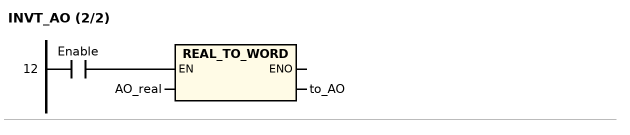
// NETWORK 12
IF Enable THEN to_AO := REAL_TO_WORD(AO_real); END_IF

END_FUNCTION_BLOCK

// Device/Application/Alarm
FUNCTION_BLOCK Alarm
VAR
	hw_alarm: STRING;
	R_DI121: R_TRIG;
	R_DI122: R_TRIG;
	R_DI123: R_TRIG;
	R_DI124: R_TRIG;
	R_DI125: R_TRIG;
	R_DI126: R_TRIG;
	R_DI127: R_TRIG;
	R_DI128: R_TRIG;
	
	B_DI121: INT;
	B_DI122: INT;
	B_DI123: INT;
	B_DI124: INT;
	B_DI125: INT;
	B_DI126: INT;
	B_DI127: INT;
	B_DI128: INT;
	
	R_DI131: R_TRIG;
	R_DI132: R_TRIG;
	R_DI133: R_TRIG;
	R_DI134: R_TRIG;
	R_DI135: R_TRIG;
	R_DI136: R_TRIG;
	R_DI137: R_TRIG;
	
	R_DI156: R_TRIG;
	
	R_DI162: R_TRIG;
	R_DI164: R_TRIG;
	R_DI166: R_TRIG;
	
	R_DI171: R_TRIG;
	R_DI172: R_TRIG;
	R_DI173: R_TRIG;
	R_DI174: R_TRIG;
	
	R_DI178: R_TRIG;
	
	R_DI181: R_TRIG;
	R_DI182: R_TRIG;
	R_DI183: R_TRIG;
	R_DI184: R_TRIG;
	R_DI185: R_TRIG;
	R_DI186: R_TRIG;
	R_DI187: R_TRIG;
	R_DI188: R_TRIG;
	
	R_DI191: R_TRIG;
	R_DI192: R_TRIG;
	R_DI193: R_TRIG;
	R_DI194: R_TRIG;
	R_DI195: R_TRIG;
	R_DI196: R_TRIG;
	
	R_DI201: R_TRIG;
	R_DI207: R_TRIG;
	R_DI208: R_TRIG;
	
	R_DI211: R_TRIG;
	
	R_DI221: R_TRIG;
	
	R_DI238: R_TRIG;
	
	R_DI241: R_TRIG;
	R_DI247: R_TRIG;
	R_DI248: R_TRIG;
	
	R_DI251: R_TRIG;
	
	alarm_ar: INT;
END_VAR

R_DI121(CLK:= DI121, Q=> );
R_DI122(CLK:= DI122, Q=> );
R_DI123(CLK:= DI123, Q=> );
R_DI124(CLK:= DI124, Q=> );
R_DI125(CLK:= DI125, Q=> );
R_DI126(CLK:= DI126, Q=> );
R_DI127(CLK:= DI127, Q=> );
R_DI128(CLK:= DI128, Q=> );
IF R_DI121.Q = TRUE AND alarm_ar < 40 THEN
	alarm_ar := alarm_ar + 1;
	hw_alarm := 'Q21 Vibrator 1 Cement Silo TRIP';
	B_DI121 := alarm_ar;
END_IF
IF R_DI122.Q = TRUE AND alarm_ar < 40 THEN
	alarm_ar := alarm_ar + 1;
	hw_alarm := 'Q23 Vibrator 2 Cement Silo TRIP';
	B_DI122 := alarm_ar; 
END_IF
IF R_DI123.Q = TRUE AND alarm_ar < 40 THEN
	alarm_ar := alarm_ar + 1;
	hw_alarm := 'Q25 Rotary Cement Silo TRIP';
	B_DI123 := alarm_ar; 
END_IF
IF R_DI124.Q = TRUE AND alarm_ar < 40 THEN
	alarm_ar := alarm_ar + 1;
	hw_alarm := 'Q27 Rotary Cement Weighter TRIP';
	B_DI124 := alarm_ar; 
END_IF
IF R_DI125.Q = TRUE AND alarm_ar < 40 THEN
	alarm_ar := alarm_ar + 1;
	hw_alarm := 'Q21 Vibrator 1 Cement Silo TRIP';
	B_DI125 := alarm_ar; 
END_IF
IF R_DI126.Q = TRUE AND alarm_ar < 40 THEN
	alarm_ar := alarm_ar + 1;
	hw_alarm := 'Q21 Vibrator 1 Cement Silo TRIP';
	B_DI126 := alarm_ar; 
END_IF
IF R_DI127.Q = TRUE AND alarm_ar < 40 THEN
	alarm_ar := alarm_ar + 1;
	hw_alarm := 'Q21 Vibrator 1 Cement Silo TRIP';
	B_DI127 := alarm_ar; 
END_IF
IF R_DI128.Q = TRUE AND alarm_ar < 40 THEN
	alarm_ar := alarm_ar + 1;
	hw_alarm := 'Q21 Vibrator 1 Cement Silo TRIP';
	B_DI128 := alarm_ar; 
END_IF

END_FUNCTION_BLOCK

// Device/Application/Constancheck
FUNCTION_BLOCK Constancheck
VAR
	ton_a: ton;
	ton_b: ton;
	catcher: r_trig;
	buffer: REAL;
	up_limit: REAL;
	down_limit: REAL;
	valid: INT;
	start_cek: BOOL;
END_VAR
VAR_INPUT
	input_value: REAL;
	tolerance: REAL := 1;
	start: BOOL;
END_VAR

VAR_OUTPUT
	output: BOOL;
END_VAR

IF start = TRUE THEN
	valid := 0;
	start_cek := TRUE;
END_IF
ton_a(IN:= NOT ton_b.Q, PT:= T#100MS, Q=> , ET=> );
ton_b(IN:= ton_a.Q, PT:= T#100MS, Q=> , ET=> );
catcher(CLK:= ton_b.Q, Q=> );
IF catcher.Q = TRUE THEN
	buffer := input_value;
	up_limit := input_value + tolerance;
	down_limit := input_value - tolerance;
	IF buffer < up_limit AND buffer > down_limit THEN
		valid := valid + 1;
		ELSE
			valid := 0;
	END_IF
END_IF
IF valid >= 25 AND start_cek = TRUE THEN
	output := TRUE;
	start_cek := FALSE;
	ELSE
		output := FALSE;
END_IF

END_FUNCTION_BLOCK

// Device/Application/DC
FUNCTION_BLOCK DC
VAR
	TON_int1: TON;
	pulse_active: BOOL;
END_VAR
VAR_OUTPUT
	tmp_int: TIME;
END_VAR
VAR
	pulse_finish: BOOL;
	CTU_0: CTU;
	TON_pulse: TON;
	TON_distance: TON;
	tmp_pulse: TIME;
	valve: INT;
	distancing: BOOL;
	tmp_dis: TIME;
END_VAR
VAR_INPUT
	pulse: TIME;
	distance: TIME;
	valve_num: INT := 6;
END_VAR
VAR
	pulsing: BOOL;
END_VAR

VAR_INPUT
	interval: TIME;
END_VAR
VAR_OUTPUT
	out_signal: WORD;
END_VAR
VAR // added by the converter: edge detectors and wires of the graphical bodies
    _rt1, _rt2, _rt3, _rt4, _rt5 : R_TRIG;
    _w1 : BOOL;
END_VAR

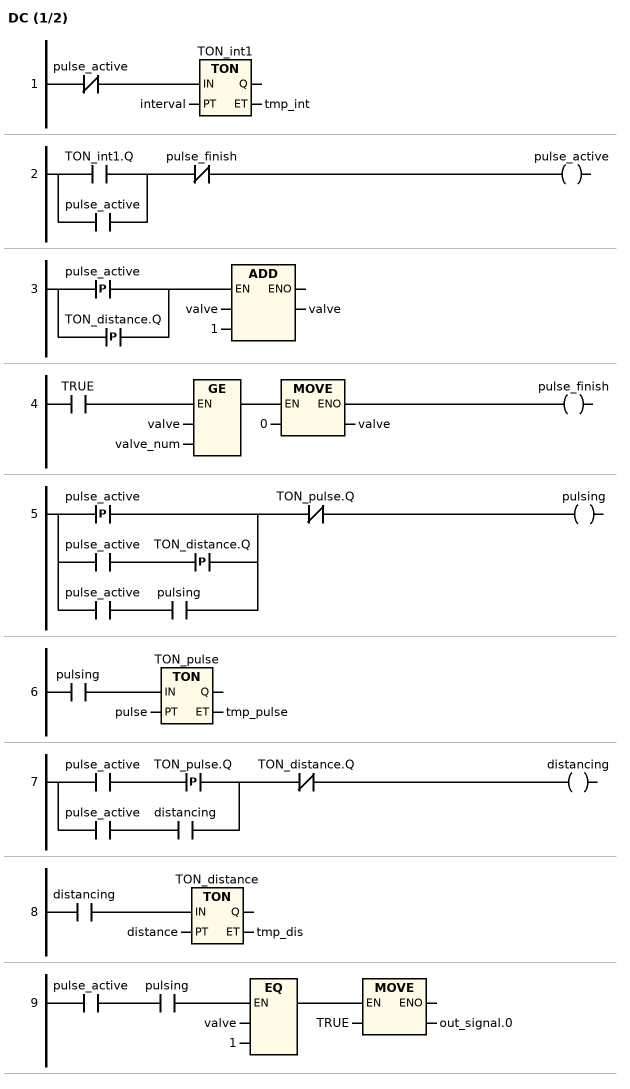
// NETWORK 1
TON_int1(IN := NOT pulse_active, PT := interval, ET => tmp_int); // TON

// NETWORK 2
pulse_active := (TON_int1.Q OR pulse_active) AND NOT pulse_finish;

// NETWORK 3
_rt1(CLK := pulse_active);
_rt2(CLK := TON_distance.Q);
IF _rt1.Q OR _rt2.Q THEN valve := valve + 1; END_IF

// NETWORK 4
_w1 := valve >= valve_num;
IF _w1 THEN valve := 0; END_IF
pulse_finish := _w1;

// NETWORK 5
_rt3(CLK := pulse_active);
_rt4(CLK := TON_distance.Q);
pulsing := (_rt3.Q OR pulse_active AND _rt4.Q OR pulse_active AND pulsing) AND NOT TON_pulse.Q;

// NETWORK 6
TON_pulse(IN := pulsing, PT := pulse, ET => tmp_pulse); // TON

// NETWORK 7
_rt5(CLK := TON_pulse.Q);
distancing := (pulse_active AND _rt5.Q OR pulse_active AND distancing) AND NOT TON_distance.Q;

// NETWORK 8
TON_distance(IN := distancing, PT := distance, ET => tmp_dis); // TON

// NETWORK 9
IF pulse_active AND pulsing AND valve = 1 THEN out_signal.0 := TRUE; END_IF

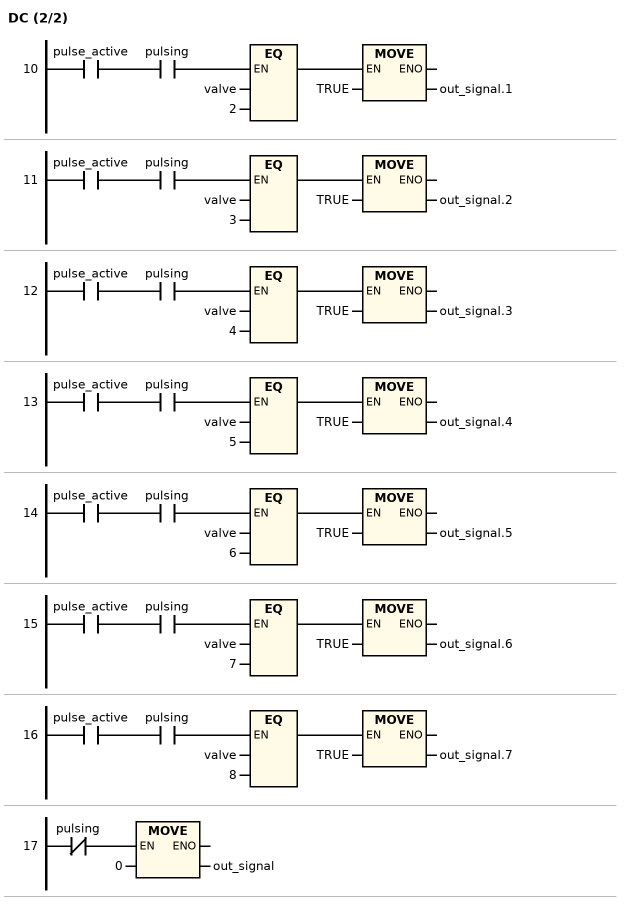
// NETWORK 10
IF pulse_active AND pulsing AND valve = 2 THEN out_signal.1 := TRUE; END_IF

// NETWORK 11
IF pulse_active AND pulsing AND valve = 3 THEN out_signal.2 := TRUE; END_IF

// NETWORK 12
IF pulse_active AND pulsing AND valve = 4 THEN out_signal.3 := TRUE; END_IF

// NETWORK 13
IF pulse_active AND pulsing AND valve = 5 THEN out_signal.4 := TRUE; END_IF

// NETWORK 14
IF pulse_active AND pulsing AND valve = 6 THEN out_signal.5 := TRUE; END_IF

// NETWORK 15
IF pulse_active AND pulsing AND valve = 7 THEN out_signal.6 := TRUE; END_IF

// NETWORK 16
IF pulse_active AND pulsing AND valve = 8 THEN out_signal.7 := TRUE; END_IF

// NETWORK 17
IF NOT pulsing THEN out_signal := 0; END_IF

END_FUNCTION_BLOCK

// Device/Application/PulseHold
FUNCTION_BLOCK PulseHold
VAR
	TON_PX : TON;
	pulse_in: BOOL;
	tmp_pulse: TIME;
	pulse_in2: BOOL;
END_VAR

VAR_INPUT
	sensor: BOOL;
	tolerance: TIME := T#5s;
	enable: BOOL;
END_VAR

VAR_OUTPUT
	output: BOOL;
END_VAR
VAR // added by the converter: edge detectors and wires of the graphical bodies
    _rt1 : R_TRIG;
    _ft1 : F_TRIG;
END_VAR

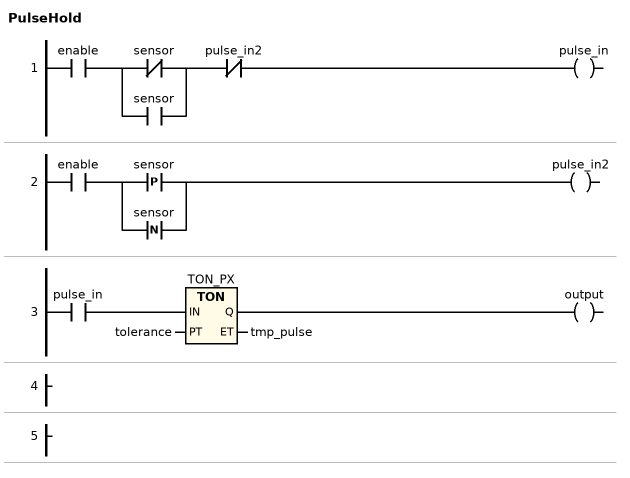
// NETWORK 1
pulse_in := enable AND (NOT sensor OR sensor) AND NOT pulse_in2;

// NETWORK 2
_rt1(CLK := sensor);
_ft1(CLK := sensor);
pulse_in2 := enable AND (_rt1.Q OR _ft1.Q);

// NETWORK 3
TON_PX(IN := pulse_in, PT := tolerance, ET => tmp_pulse); // TON
output := TON_PX.Q;

// NETWORK 4

// NETWORK 5

END_FUNCTION_BLOCK

// Device/Application/Logger
PROGRAM Logger
VAR
	oMySql : MySQL_Context; (* Used like Structure for keeping login and status information - Do not call it within your program *)
	
	
	(* Functionblock to contact MySql server *)
	
	oLogin : MYSQL_Login;
	xConnect : BOOL;
	diErrorLogin : DINT;
	sStatusLogin : STRING(200);
	xConnected : BOOL;

	(* Functionblock to process SQL statements who do not return result sets *)
	oExec1 : MYSQL_Execute;
	asSqlStatement1 : ARRAY [0..gcMySql_iSqlUpperBound] OF STRING(gcMySQL_iSqlLength);
	xExec1 : BOOL;
	diErrorExec1 : DINT;
	sStatusExec1 : STRING(200);

	(* Functionblock to process SQL statements who return result sets *)
	oQuery2 : MySQL_Query;
	asSqlStatement2 : ARRAY [0..gcMySql_iSqlUpperBound] OF STRING(gcMySQL_iSqlLength);
	xQuery2 : BOOL;
	diErrorQuery2 : DINT;
	sStatusQuery2 : STRING(200);
	stResultSet :MySQL_ResultSet;

	(* Functionblock to disconnect from MSSQL server *)
	oLogout : MySQL_Logout;
	xDisconnect : BOOL;
	diErrorLogout : DINT;
	sStatusLogout : STRING(200);

	
	TON_CONNECT: TON;
	
	TOF_RESETER: TOF;
	reseting: BOOL;
	res: R_TRIG;
END_VAR

TON_CONNECT( IN := NOT xConnected, PT := T#10S);
 
IF TON_CONNect.Q THEN 
	TON_CONNECT( IN := FALSE, PT := T#10S);
	xConnect := TRUE;
END_IF


oLogin(
	sHost:= '192.168.1.11', 
	uiPort:= 3306, 
	sUsername:= 'nodejs', 
	sPassword:= 'nodejs', 
	//sAppName:= , 
	//sLibName:= , 
	sDatabase:= 'db_codesys', 
	oMySql:= oMySql, 
	xStart:= xConnect, 
	diError=> diErrorLogin, 
	sStatus=> sStatusLogin, 
	xConnected=> xConnected);
	
	IF xConnected THEN
		IF Automode.log_mortar THEN 
			asSqlStatement1[0] := 'call mor(';
			asSqlStatement1[0] := CONCAT(asSqlStatement1[0], INT_TO_STRING(0));
			asSqlStatement1[0] := CONCAT(asSqlStatement1[0], ',"');
			asSqlStatement1[0] := CONCAT(asSqlStatement1[0], Formula.formula_name);
			asSqlStatement1[0] := CONCAT(asSqlStatement1[0], '",');
			asSqlStatement1[0] := CONCAT(asSqlStatement1[0], REAL_TO_STRING(Formula.cement_target));
			asSqlStatement1[0] := CONCAT(asSqlStatement1[0], ',');
			asSqlStatement1[0] := CONCAT(asSqlStatement1[0], REAL_TO_STRING(Formula.lime_target));
			asSqlStatement1[0] := CONCAT(asSqlStatement1[0], ',');
			asSqlStatement1[0] := CONCAT(asSqlStatement1[0], REAL_TO_STRING(Formula.sand_target));
			asSqlStatement1[0] := CONCAT(asSqlStatement1[0], ',');
			asSqlStatement1[0] := CONCAT(asSqlStatement1[0], REAL_TO_STRING(Automode.start_cement));
			asSqlStatement1[0] := CONCAT(asSqlStatement1[0], ',');
			asSqlStatement1[0] := CONCAT(asSqlStatement1[0], REAL_TO_STRING(Automode.end_cement));
			asSqlStatement1[0] := CONCAT(asSqlStatement1[0], ',');
			asSqlStatement1[0] := CONCAT(asSqlStatement1[0], INT_TO_STRING(Automode.weighting_duration));
			asSqlStatement1[0] := CONCAT(asSqlStatement1[0], ',');
			asSqlStatement1[0] := CONCAT(asSqlStatement1[0], REAL_TO_STRING(LimeSand.start_lime));
			asSqlStatement1[0] := CONCAT(asSqlStatement1[0], ',');
			asSqlStatement1[0] := CONCAT(asSqlStatement1[0], REAL_TO_STRING(LimeSand.end_lime));
			asSqlStatement1[0] := CONCAT(asSqlStatement1[0], ',');
			asSqlStatement1[0] := CONCAT(asSqlStatement1[0], INT_TO_STRING(LimeSand.weighting_duration));
			asSqlStatement1[0] := CONCAT(asSqlStatement1[0], ',');
			asSqlStatement1[0] := CONCAT(asSqlStatement1[0], REAL_TO_STRING(Cement_PRG.start_cement_dosing));
			asSqlStatement1[0] := CONCAT(asSqlStatement1[0], ',');
			asSqlStatement1[0] := CONCAT(asSqlStatement1[0], REAL_TO_STRING(Cement_PRG.end_cement_dosing));
			asSqlStatement1[0] := CONCAT(asSqlStatement1[0], ',');
			asSqlStatement1[0] := CONCAT(asSqlStatement1[0], INT_TO_STRING(Cement_PRG.dosing_duration));
			asSqlStatement1[0] := CONCAT(asSqlStatement1[0], ')');
			xExec1 := TRUE;
		END_IF
		IF LimeSand.finish_button THEN 
			asSqlStatement1[0] := 'INSERT INTO mo_lime(val, frm, act) VALUES(';
			asSqlStatement1[0] := CONCAT(asSqlStatement1[0], REAL_TO_STRING(LimeSand.lime_progress));
			asSqlStatement1[0] := CONCAT(asSqlStatement1[0], ',');
			asSqlStatement1[0] := CONCAT(asSqlStatement1[0], REAL_TO_STRING(Formula.lime_target));
			asSqlStatement1[0] := CONCAT(asSqlStatement1[0], ',');
			asSqlStatement1[0] := CONCAT(asSqlStatement1[0], REAL_TO_STRING(LimeSand.lime_weight));
			asSqlStatement1[0] := CONCAT(asSqlStatement1[0], ')');
			xExec1 := TRUE;
		END_IF
		IF Cement_PRG.log_cem THEN 
			asSqlStatement1[0] := 'INSERT INTO mo_cem(val, frm) VALUES(';
			asSqlStatement1[0] := CONCAT(asSqlStatement1[0], REAL_TO_STRING(Cement_PRG.cement_weight));
			asSqlStatement1[0] := CONCAT(asSqlStatement1[0], ',');
			asSqlStatement1[0] := CONCAT(asSqlStatement1[0], REAL_TO_STRING(formula.cement_target));
			asSqlStatement1[0] := CONCAT(asSqlStatement1[0], ')');
			xExec1 := TRUE;
		END_IF
		IF Automode.TON_4.Q THEN 
			asSqlStatement1[0] := 'INSERT INTO mo_clk(val) VALUES(';
			asSqlStatement1[0] := CONCAT(asSqlStatement1[0], '1');
			asSqlStatement1[0] := CONCAT(asSqlStatement1[0], ')');
			xExec1 := TRUE;
		END_IF
	END_IF
	
	
	oExec1(
	asSqlCommand:= asSqlStatement1, 
	oMySql:= oMySql, 
	xStart:= xExec1, 
	diError=> diErrorExec1, 
	sStatus=> sStatusExec1);
	
	IF diErrorExec1 <> 0 THEN
		reseting := TRUE;
	END_IF
	res(CLK:= reseting, Q=> );
	TOF_RESETER(IN:= res.Q, PT:= T#3S, Q=> , ET=> );

END_PROGRAM

// Device/Application/MYSQL/private/MySql_Context
FUNCTION_BLOCK MySql_Context
(*  This function block is used like a STRUCT for keeping login and status informations.
	
	Define one instance of this function block in your plc program and use it only as 
	input param for all the other function blocks of this library.

	Do not "call" this functionblock inside your plc program.

	In addition this function block provide the one and only receive and transmit buffer 
	for this library and operate as schedular for function blocks who want to talk with 
	the database server.
 *)
VAR_INPUT
  	sHost : STRING;		  	(* IP or hostname where MySQL-server is working *)
  	uiPort : UINT;			(* TCP-Port where MySQL-server is listening, typ. 3306 *)
	sUsername : STRING;
	sPassword : STRING;
	sDatabase : STRING;	  	(* Name of schema to use initially - Optional param*)

	stServerInfo : MySql_ServerInfo; (* See structure "MySql_ServerInfo" for details *)

	xConnected : BOOL; (* Succesful logged into database *)

	(*- Private ----------------------------------------------*)
	(* The one and only socket handle *)
	dwSocketHandle : DWORD; (* Handle for Read/Write data *)
	(* The one and only transmit buffer *)
	abTxBuffer	   : ARRAY[0..gcMySql_dwTxBufferSize] OF BYTE;
	(* The one and only receive buffer *)
	abRxBuffer	   : ARRAY[0..gcMySql_dwRxBufferSize] OF BYTE;
	(* The one and only semaphore to synchronize buffer access *)
	dwBufferSemaphor : DWORD; (* Handle to semaphore *)

END_VAR
VAR_OUTPUT
END_VAR
VAR

END_VAR

;

END_FUNCTION_BLOCK

// Device/Application/MYSQL/public/MySql_Login
FUNCTION_BLOCK MySql_Login
(* This function is used to connect to a MySQL-Server

	RetVal dwError:	
		16#00000000 => 'SUCCESS'
		16#80001001 => 'TCP-ERROR: DNS-Request failed, could not retrieve servers IP address'
		16#80001002 => 'TCP-ERROR: Could not convert servers IP address into dotted format'
		16#80001003 => 'TCP-ERROR: "SysSockCreate()" fails - Could not get socket'
		16#80001004 => 'TCP-ERROR: Switching to none blocking mode fails'
		16#80001005 => 'TCP-ERROR: "SysSockRecv()" returns 0. Socket was "gracefully closed"'
		16#80001006 => 'TCP-ERROR: "SysSockSend()" returns 0. Socket was "gracefully closed"'
		16#80001007 => 'TCP-ERROR: "SysSockSend()" returns -1'
		16#80004001 => 'PARAM-ERROR: ' 
		16#80004002 => 'PARAM-ERROR: "MySql.sHost" not assigned' 
		16#80004003 => 'PARAM-ERROR: "MySql.sUser" not assigned' 
		16#80005001 => 'MYSQL-ERROR: Library requires protocol version 10 or above. Server support only version x' 
		16#80005002 => 'MYSQL-ERROR: <Message from server>	
		16#80005003 => 'MYSQL-ERROR: Invalid or unexpected response from server'
		16#80005004 => 'MYSQL-ERROR: Function "MySql_Scramble()" returns with error'

		16#80004001 => 'TIMEOUT: <actual processed step in state machine>'

	ToDo's: 
		- Add checks for Server-Status and Server-Capabilties in "wState=35"

 date     | release	| author  | Desc
----------+---------+------------------------------------------------------------
 24.01.12 |  3.4	| CM      | Bugfix - Set PUSH-Bit also for 88x controllers 
 29.09.10 |  2.4    | CM      | Bugfix for IP in dotted format
 28.09.10 |  2.3    | CM      | Add DNS support for 750-881 and derivates
 28.09.10 |  2.2    | CM      | Add error message when Login not allowed for this host
 06.08.10 |  2.0	| CM      | Init 
*)
VAR_INPUT
  	sHost	  : STRING; 	 (* IP or hostname where MySQL-server is working *)
  	uiPort 	  : UINT := 3306;(* TCP-Port where MySQL-server is listening, typ. 3306 *)
	sUsername : STRING;		 (* Name of database account *)
	sPassword : STRING;   	 (* Password of database account *)
	sDatabase : STRING;	     (* Name of schema to use initially - Optional param*)
END_VAR
VAR_IN_OUT
	oMySql : MySql_Context;  (* Structure for keeping login and status informations *)
	xStart : BOOL; 			 (* Start execution on a rising edge and reset internally when done or on timeout.  *)
END_VAR
VAR_OUTPUT
	diError : DWORD; 		 (* Numeric return value - more readable in hex  *)
	sStatus : STRING(200); 	 (* Textual description of current state or error *)
	xConnected : BOOL;		 (* TRUE: when database connection is established *)
END_VAR
VAR
	wState : WORD;	 (* State mashine *)

	oTON			: TON;		(* Watchdogtimer for statemashine *)

	xWatchDogOn		: BOOL; 	(* enable disable Watchdog for statemashine *)
	wStateOld		: WORD;		(* persist the last state of statemashine *)

	sServerIpDotted	: STRING; 	(* Ip-Adress in dottet format '192.168.1.12' *)
	dwServerIp		: DWORD;	(* Ip-Adress in DWORD format  16#C0A8010C *)
	oInAddr	  		: INADDR;  	(* IP-Address as DWORD*)
	stSockAddr		: SOCKADDRESS;
	c_fdWrite : SOCKET_FD_SET;
	c_Timeout : SOCKET_TIMEVAL;

	dwSocket 	 	: DWORD; (* Socket handle *)
	diTcpOption  	: DINT := 1;
	diIoCtlParam 	: DINT := 1; (* IOCTL-Parameter for non-blocking mode of sockets *)
	xResult		 	: BOOL;		(* Return value of functions *)
	diResult		: __XINT; 	(* Retval value of functions *)

	diTxCount		: __XINT; (* Number of bytes to send *)
	diRxCount		: __XINT; (* Number of received bytes *)

	(* Local Buffer *)
	abToken : ARRAY[0..20] OF BYTE;  (* "abToken" calculatet from "salt" and "password" for login, when "password" is assigned *)

	(* Helpers *)
	dwPacketLength : DWORD; (*  *)
	uiPos : UINT;
	wMask : WORD := 16#00FF;
	dwMask : DWORD := 16#000000FF;

	i : INT;
	iHelp : INT;
	psHelp : POINTER TO STRING(180);
	pabHelp : POINTER TO ARRAY [0..512] OF BYTE;
	c_select: BOOL;
	RTS_IEC_RES: UDINT;
	ptrDINT : POINTER TO DINT;
	Sock_Host : SOCK_HOSTENT;
	Ready: INT;
	pIPAddress: POINTER TO DWORD;
END_VAR

CASE  wState OF (* The state maschine *********************************************)

0:	(* Idle - wait for something to do -------------------------------------------*)
	IF xStart THEN
		diError := 0;
		sStatus := '';
		MySql_Close(oMySql); (* Kill existing connection when user login two times *)
		oMySql.xConnected := FALSE;
		xConnected := oMySql.xConnected;
		wState := 5; (* Go ahead *)
	END_IF

5: (* Check structure "oMySql" for valid values *)
	IF sHost <> '' THEN
		oMySql.sHost := sHost;
	ELSE
		diError := 16#80004002;
		sStatus :='PARAM-ERROR: "sHost" not assigned';
		wState:=999;
		RETURN; (* ---- RETURN -----*)
	END_IF
	IF sUsername <> '' THEN
		oMySql.sUsername := sUsername;
	ELSE
		diError := 16#80004003;
		sStatus :='PARAM-ERROR: "sUsername" not assigned';
		wState:=999;
		RETURN; (* ---- RETURN -----*)
	END_IF
	oMySql.uiPort := uiPort;
	oMySql.sPassword := sPassword;
	oMySql.sDatabase := sDatabase;
	wState := 10; (* Go ahead *)

10:	(* Check if given address is "hostname" or "IP address in dottet format" --------------*)
	RTS_IEC_RES := SysSockInetAddr(oMySql.sHost, ADR(dwServerIp));
	IF RTS_IEC_RES = 16#00000000 AND dwServerIp <> 16#00000000 THEN
		sServerIpDotted:=oMySql.sHost;
		oInAddr.ulAddr := dwServerIp;
		wState:=15; 	(*Input is already the IP address in dottet format*)
	ELSE
		wState:=12; 	(*Input is a hostname *)
	END_IF

12: (* Send a DNS-Request to obtain servers IP address for the given hostname --------------*)
	RTS_IEC_RES := SysSockGetHostByName(oMySql.sHost,ADR(Sock_Host));
	pIPAddress := Sock_Host.pAddrList[0];
	dwServerIp := pIPAddress^;
	IF dwServerIp <> SOCKET_INADDR_NONE THEN
		wState:=14;
	ELSE
		diError := 16#80001001;
		sStatus :='TCP-ERROR: DNS-Request failed, could not retrieve servers IP address';
		wState:=999;
	END_IF

14: (* Convert Ip address from DWORD into dotted format ------------------------------------*)
(* Change byteorder from network to host order *)
	(*CASE ADR(%MW0) OF
	16#30000000 : (* For 750-841 *)
		oInAddr.S_addr:=SysSockNtohl(dwNet:=dwServerIp); (* Change byteorder from network to host order *)
	16#20000000 : (* For 750-881 *)
		oInAddr.S_addr:=SysSockNtohl(dwNet:=dwServerIp); (* Change byteorder from network to host order *)
	ELSE
		(* For 758-870 *)
		oInAddr.S_addr:= dwServerIp; (* Byteorder allready ok *)
	END_CASE*)
	oInAddr.ulAddr := dwServerIp; (* Byteorder allready ok *)
	RTS_IEC_RES := SysSockInetNtoa(pInAddr:=ADR(oInAddr), szIPAddr:= sServerIpDotted, diIPAddrSize:= SIZEOF(sServerIpDotted));
	xResult := (RTS_IEC_RES = 0);
	IF xResult THEN
		wState:=15;
	ELSE
		diError := 16#80001002;
		sStatus :='TCP-ERROR: Could not convert servers IP address into dotted format';
		wState:=999;
	END_IF

15: (* Create socket descriptor  ---------------------------*)
	(*dwSocket := SysSockCreate(diAddressFamily := SOCKET_AF_INET,
							  diType		  := SOCKET_STREAM,
							  diProtocol 	  := SOCKET_IPPROTO_IP);*)
	dwSocket := SysSockCreate(						 iAddressFamily	:= SOCKET_AF_INET,
													 diType		:= SOCKET_STREAM,
													 diProtocol := SOCKET_IPPROTO_TCP,
													 pResult := ADR(RTS_IEC_RES));
	IF dwSocket >= 0 THEN
		oMySql.dwSocketHandle := dwSocket;  (* Make handle available for other function blocks *)
		(* Set Push-Bit only for 750-841 and derivates *)
		IF TRUE THEN (*((ADR(%MW0)=16#30000000) OR (ADR(%MW0)=16#20000000)) THEN (*841, 871, 872, 873, 880 ... *)*)
			(*SysSockSetOption(diSocket		:= dwSocket,
							 diLevel		:= 6,
							 diOption		:= SOCKET_TCP_NODELAY,
							 pOptionValue	:= ADR(),
							 diOptionLength	:= SIZEOF(diTcpOption));*)
			SysSockSetOption(
						hSocket:=dwSocket,
						diLevel:=6,
						diOption:=SOCKET_TCP_NODELAY,
						pdiOptionValue:=ADR(diTcpOption),
						diOptionLen:=SIZEOF(diTcpOption));
		END_IF
		wState := 16; (* Go ahead *)
	ELSE
		diError := 16#80001003;
		sStatus :='TCP-ERROR: "SysSockCreate()" fails - Could not get socket';
		wState:=999;
	END_IF

16: (* Change socket mode to "nonblocking" ---------------------------*)
	diResult := SysSockIoctl( dwSocket,
							  SOCKET_FIONBIO,
							  ADR(diIoCtlParam));
	IF TRUE THEN (*diResult <> 0 THEN*)
		stSockAddr.sin_family := SOCKET_AF_INET;
		stSockAddr.sin_port := SysSockNtohs(uiPort);
		stSockAddr.sin_addr.ulAddr := oInAddr.ulAddr;
		sStatus := CONCAT('Try to connect with ', oMySql.sHost);
		wState := 18;
	ELSE
		diError := 16#80001004;
		sStatus :='TCP-ERROR: Switching to none blocking mode fails';
		wState:=999;
	END_IF

18: (* Create and occupy semaphore to synchronize buffer handling for socket operations *)
	oMySql.dwBufferSemaphor := SysSemCreate(ADR(RTS_IEC_RES)); (* Create semaphore  *)
	SysSemEnter(oMySql.dwBufferSemaphor); (* CAUTION: SysSemEnter() is a blocking function *)
	c_select := FALSE;
	wState := 20;

20: (* Connect with server ---------------------------*)
	sStatus :=CONCAT('Try to connect to ', oMySql.sHost);
	IF c_select = FALSE THEN
			RTS_IEC_RES := SysSockConnect( dwSocket, ADR(stSockAddr),  SIZEOF(stSockAddr));
			xResult := (RTS_IEC_RES = 0);
			IF NOT xResult THEN
						sStatus :='Connection established - Waiting for "Handshake Initialisation Packet" from server';
						wState:=25;
			ELSE
					c_select := TRUE;
			END_IF
	ELSE
			c_Timeout.tv_sec := 0;
			c_Timeout.tv_usec := 0;
			c_fdWrite.fd_count := 1;
			c_fdWrite.fd_array[0] := dwSocket;
			SysSockSelect(SOCKET_FD_SETSIZE,0,ADR(c_fdWrite),0, ADR(c_Timeout), ADR(Ready));
			xResult := Ready > 0;
			IF xResult THEN (* succesful *)
				sStatus :='Connection established - Waiting for "Handshake Initialisation Packet" from server';
				wState:=25;
			END_IF
	END_IF
25: (* Read "Handshake Initialisation Packet" received from server *)
	(*diRxCount := SysSockRecv(diSocket 	:= dwSocket,
							 pbyBuffer 	:= ADR(oMySql.abRxBuffer),		(* Address of receive buffer *)
							 diBufferSize:= SIZEOF(oMySql.abRxBuffer),
							 diFlags	:= 0);*)
		diRxCount := SysSockRecv(		hSocket 	:= dwSocket,
										pbyBuffer 	:= ADR(oMySql.abRxBuffer),		(* Address of receive buffer *)
										diBufferSize:= SIZEOF(oMySql.abRxBuffer),
										diFlags		:= 0,
										pResult := ADR(RTS_IEC_RES));						 

	CASE diRxCount OF
	-1:(* No data available or error occured *)
			; (* Let the watchdog look for *)

	(*0: (* Socket was "gracefully closed"  *)*)
		diError := 16#80001005;
		sStatus :='TCP-ERROR: "SysSockRecv()" returns 0. Socket was "gracefully closed"';
		wState:=999;

	ELSE (* We receive some data from server *)
		IF RTS_IEC_RES <> 0 AND RTS_IEC_RES <> 518 THEN
			diError := 16#80001005;
			sStatus :='TCP-ERROR: "SysSockRecv()" returns 0. Socket was "gracefully closed"';
			wState:=999;
		ELSE
		IF diRxCount > 0 THEN
		dwPacketLength := 	BYTE_TO_DWORD(oMySql.abRxBuffer[0]) OR
							SHL(BYTE_TO_DWORD(oMySql.abRxBuffer[1]),8) OR
							SHL(BYTE_TO_DWORD(oMySql.abRxBuffer[2]),16);
		IF diRxCount >= dwPacketLength THEN
			wState:=27; (* Go ahead *)
		END_IF
		END_IF
		END_IF
	END_CASE

27: (* Check if response a "Handshake Initialisation Packet" *)
	IF oMySql.abRxBuffer[4] = 16#FF THEN
		(* Error frame received - Copy error message *)
		psHelp := ADR(oMySql.abRxBuffer[7]);
		diError := 16#80005002;
		sStatus := CONCAT('MYSQL-ERROR: ', psHelp^);
		wState:=999;
	ELSE
		sStatus :='"Handshake Initialisation Packet" received - Generate "Scramble-Key"';
		wState:=30; (* Go ahead *)
	END_IF

30:	(* Copy informations from "server greetings" into context "oMySql.stServerInfo" *)
	(* Copy "Protocol-Version" to context *)
	oMySql.stServerInfo.bProtocolVersion := oMySql.abRxBuffer[4];
	(* Copy "Server-Version" to context *)
	psHelp := ADR(oMySql.abRxBuffer[5]);
	oMySql.stServerInfo.sServerVersion := psHelp^;
	(* Calculate Posion of Thread-Id in receive buffer *)
	uiPos := 5 +LEN(psHelp^)+1;
	(* Copy "Thread-Id"(4Byte) to context *)
	oMySql.stServerInfo.dwThreadId :=    BYTE_TO_DWORD(oMySql.abRxBuffer[uiPos])       OR
										SHL(BYTE_TO_DWORD(oMySql.abRxBuffer[uiPos+1]),8)  OR
										SHL(BYTE_TO_DWORD(oMySql.abRxBuffer[uiPos+2]),16) OR
										SHL(BYTE_TO_DWORD(oMySql.abRxBuffer[uiPos+3]),24);
	uiPos := uiPos +4;
	(* Copy first part (8Byte) of "Scramble-Buffer" to context *)
	FOR i:=0 TO 7 DO
		oMySql.stServerInfo.abScrambleBuffer[i] := oMySql.abRxBuffer[uiPos+i];
	END_FOR
	uiPos := uiPos +8 +1;
	(* Copy "Server-Capabilities" to context *)
	oMySql.stServerInfo.wServerCapabilities := 	BYTE_TO_WORD(oMySql.abRxBuffer[uiPos])       OR
												SHL(BYTE_TO_WORD(oMySql.abRxBuffer[uiPos+1]),8);
	uiPos := uiPos +2;
	(* Copy "Server-Language" to context *)
	oMySql.stServerInfo.bServerLanguageId := oMySql.abRxBuffer[uiPos];
	uiPos := uiPos +1;
	(* Copy "Server-Status" to context *)
	oMySql.stServerInfo.wServerStatus := BYTE_TO_WORD(oMySql.abRxBuffer[uiPos])       OR
										SHL(BYTE_TO_WORD(oMySql.abRxBuffer[uiPos+1]),8);
	uiPos := uiPos +2+13;
	(* Copy rest(13Byte) of "Scramble-Buffer" to context *)
	FOR i:=0 TO 12 DO
		oMySql.stServerInfo.abScrambleBuffer[8 +i] := oMySql.abRxBuffer[uiPos+i];
	END_FOR
	wState:=35;

35: (* Check informations from "server greetings" *)
	IF oMySql.stServerInfo.bProtocolVersion < 10 THEN
		diError := 16#80005001;
		sStatus :=CONCAT('MYSQL-ERROR: Library requires protocol version 10 or above. Server support only version ', BYTE_TO_STRING(oMySql.stServerInfo.bProtocolVersion));
		wState:=999;
		RETURN;
	END_IF
	wState:=40;

40: (* Calculate "Token" for login from "salt" and "password", when "password" is assigned *)
	IF oMySql.sPassword = '' THEN
		wState:=45;
	ELSE
		xResult := MySql_Scramble(oMySql.stServerInfo.abScrambleBuffer,
								  oMySql.sPassword,
							      abToken);
		IF xResult THEN
			wState:=45;
		ELSE
			diError := 16#80005004;
			sStatus :='MYSQL-ERROR: Function "MySql_Scramble()" returns with error';
			wState:=999;
		END_IF
	END_IF

45: (* Prepare "Client Authentication Packet" or "Login Request" ---------------------------*)
	(* Packet-Length - will be calculated and assigned at the end of this step *)
	oMySql.abTxBuffer[ 0] := 16#00;
	oMySql.abTxBuffer[ 1] := 16#00;
	oMySql.abTxBuffer[ 2] := 16#00;
	(* Packet-Number *)
	oMySql.abTxBuffer[ 3] := 1;
	(* Client-Capabilties *)
	oMySql.abTxBuffer[ 4] := WORD_TO_BYTE(gcMySql_wClientFlags AND wMask);
	oMySql.abTxBuffer[ 5] := WORD_TO_BYTE(SHR(gcMySql_wClientFlags, 8) AND wMask);
	(* Client-Capabilties - Extended *)
	oMySql.abTxBuffer[ 6] := WORD_TO_BYTE(gcMySql_wExtClientFlags AND wMask);
	oMySql.abTxBuffer[ 7] := WORD_TO_BYTE(SHR(gcMySql_wExtClientFlags, 8) AND wMask);
	(* Max-Packet-Size *)
	oMySql.abTxBuffer[ 8] := DWORD_TO_BYTE(gcMySql_dwMaxPacketSize AND dwMask);
	oMySql.abTxBuffer[ 9] := DWORD_TO_BYTE(SHR(gcMySql_dwMaxPacketSize, 8) AND dwMask);
	oMySql.abTxBuffer[10] := DWORD_TO_BYTE(SHR(gcMySql_dwMaxPacketSize, 16) AND dwMask);
	oMySql.abTxBuffer[11] := DWORD_TO_BYTE(SHR(gcMySql_dwMaxPacketSize, 24) AND dwMask);
	(* Character-Set *)
	oMySql.abTxBuffer[12] := gcMySql_bCharsetNumber;
	(* Filler - 23 byte allways 16#00 *)
	FOR i:=0 TO 22 DO
		oMySql.abTxBuffer[13+i] := 16#00;
	END_FOR
	uiPos := 13 + 23;
	(* Username (Null-Terminated String) *)
	pabHelp := ADR(sUsername);
	iHelp := LEN(sUsername);
	FOR i:=0 TO iHelp DO
		oMySql.abTxBuffer[uiPos+i] := pabHelp^[i];
	END_FOR
	uiPos := uiPos + iHelp +1;
	(* When Password is given *)
	IF sPassword = '' THEN
		(* Password (Length Coded Binary) *)
		oMySql.abTxBuffer[uiPos] := 16#00; (* Length *)
		uiPos := uiPos +1;
	ELSE
		(* Password (Length Coded Binary) *)
		oMySql.abTxBuffer[uiPos] := 20; (* Length *)
		uiPos := uiPos +1;
		(* Scrambled-Key *)
		FOR i:=0 TO 20 DO
			oMySql.abTxBuffer[uiPos+i] := abToken[i];
		END_FOR
		uiPos := uiPos +20;
	END_IF

	(* Calculate number of bytes to transmit and logical packet-length *)
	diTxCount := uiPos; (* Bytes to send *)
	dwPacketLength := uiPos -4;

	(* Packet-Length *)
	oMySql.abTxBuffer[ 0] := DWORD_TO_BYTE(dwPacketLength AND dwMask);
	oMySql.abTxBuffer[ 1] := DWORD_TO_BYTE(SHR(dwPacketLength, 8) AND dwMask);
	oMySql.abTxBuffer[ 2] := DWORD_TO_BYTE(SHR(dwPacketLength, 16) AND dwMask);
	sStatus :='Send "Login Request Packet" to server';
	wState := 50;

50: (* Send "Client Authentication Packet*)
	(*diResult := SysSockSend(diSocket := dwSocket,
							pbyBuffer := ADR(oMySql.abTxBuffer),
							diBufferSize := diTxCount,
							diFlags := 0);*)
	diResult := SysSockSend(	hSocket := dwSocket,
								pbyBuffer := ADR(oMySql.abTxBuffer),
								diBufferSize := diTxCount,
								diFlags := 0,
								pResult := ADR(RTS_IEC_RES));

	CASE diResult OF
	-1:	(* ERROR *)
		diError := 16#80001007;
		sStatus :='TCP-ERROR: "SysSockSend()" returns -1';
		wState:=999;
	0: (* Socket was "gracefully closed" *)
		diError := 16#80001007;
		sStatus :='TCP-ERROR: "SysSockSend()" returns 0. Socket was "gracefully closed"';
		wState:=999;
	ELSE (* succesful *)
		sStatus :='Waiting for "OK Packet" from server';
		wState:=55;
	END_CASE

55: (* Wait for "Response" from server *)
	(*diRxCount := SysSockRecv(diSocket 	:= dwSocket,
							 pbyBuffer 	:= ADR(oMySql.abRxBuffer),		(* Address of receive buffer *)
							 diBufferSize:= SIZEOF(oMySql.abRxBuffer),
							 diFlags	:= 0);*)
	diRxCount := SysSockRecv(		hSocket 	:= dwSocket,
										pbyBuffer 	:= ADR(oMySql.abRxBuffer),		(* Address of receive buffer *)
										diBufferSize:= SIZEOF(oMySql.abRxBuffer),
										diFlags		:= 0,
										pResult := ADR(RTS_IEC_RES));
	CASE diRxCount OF
	-1:(* No data available or error occured *)
			; (* Let the watchdog look for *)

	(*0: (* Socket was "gracefully closed"  *)*)
		diError := 16#80001005;
		sStatus :='TCP-ERROR: "SysSockRecv()" returns 0. Socket was "gracefully closed"';
		wState:=999;

	ELSE (* We receive some data from server *)
		IF RTS_IEC_RES <> 0 AND RTS_IEC_RES <> 518 THEN
			diError := 16#80001005;
			sStatus :='TCP-ERROR: "SysSockRecv()" returns 0. Socket was "gracefully closed"';
			wState:=999;
		ELSE
		IF diRxCount > 0 THEN
		dwPacketLength := 	BYTE_TO_DWORD(oMySql.abRxBuffer[0]) OR
							SHL(BYTE_TO_DWORD(oMySql.abRxBuffer[1]),8) OR
							SHL(BYTE_TO_DWORD(oMySql.abRxBuffer[2]),16);
		IF diRxCount >= dwPacketLength THEN
			wState:=60; (* Go ahead *)
		END_IF
		END_IF
		END_IF
	END_CASE

60: (* Check response packet, could be OK- or ERROR-Packet *)
	CASE oMySql.abRxBuffer[4] OF (* field "field_count"*)

	16#00: (* OK-Packet: Identified by "field_count", always = 0 *)
		IF sDatabase <> '' THEN
			(* Send "COM_INIT_DB" command to select specified database *)
			wState:=65;
		ELSE
			(* Everything fine - nothing else to do *)
			wState:=90;
		END_IF


	16#FF: (* ERROR-Packet: Identified by "field_count", always = 16#FF *)
		diError := 16#80005002;
		(* Copy server message into "sStatus"*)
		sStatus :='MYSQL-ERROR:  ';
		pabHelp := ADR(sStatus)+13;
		FOR i:=0 TO DWORD_TO_INT(dwPacketLength-10) DO
			pabHelp^[i] := oMySql.abRxBuffer[13+i];
			IF i>=499 THEN
				EXIT;
			END_IF
		END_FOR
		pabHelp^[i] := 16#00;
		wState:=999;

	ELSE (* Invalid or unexpected response from server (at this time) *)
		diError := 16#80005003;
		sStatus :='MYSQL-ERROR: Invalid or unexpected response from server';
		wState:=999;
	END_CASE

65: (* Prepare "COM_INIT_DB" command to select specified database *)
	(* Calculate Packet-Length *)
	iHelp := LEN(sDatabase); (* argument *)
	dwPacketLength := 1 + iHelp; (* command + argument *)
	diTxCount := dwPacketLength +4; (* Bytes to send (command + argument + header) *)
	(* Packet-Length *)
	oMySql.abTxBuffer[0] := DWORD_TO_BYTE(dwPacketLength AND dwMask);
	oMySql.abTxBuffer[1] := DWORD_TO_BYTE(SHR(dwPacketLength, 8) AND dwMask);
	oMySql.abTxBuffer[2] := DWORD_TO_BYTE(SHR(dwPacketLength, 16) AND dwMask);
	(* Packet-Number *)
	oMySql.abTxBuffer[3] := 0;
	(* Command *)
	oMySql.abTxBuffer[4] := 16#02; (* "COM_INIT_DB" command *)
	(* Argument *)
	pabHelp := ADR(sDatabase);
	FOR i:=0 TO iHelp-1 DO
		oMySql.abTxBuffer[5+i] := pabHelp^[i];
	END_FOR
 	(* Send "COM_INIT_DB" command to select specified database *)
	(*diResult := SysSockSend(diSocket := dwSocket,
							pbyBuffer := ADR(oMySql.abTxBuffer),
							diBufferSize := diTxCount,
							diFlags := 0);*)
	diResult := SysSockSend(	hSocket := dwSocket,
								pbyBuffer := ADR(oMySql.abTxBuffer),
								diBufferSize := diTxCount,
								diFlags := 0,
								pResult := ADR(RTS_IEC_RES));
							
	CASE diResult OF
	-1:	(* ERROR *)
		diError := 16#80001007;
		sStatus :='TCP-ERROR: "SysSockSend()" returns -1';
		wState:=999;
	0: (* Socket was "gracefully closed" *)
		diError := 16#80001007;
		sStatus :='TCP-ERROR: "SysSockSend()" returns 0. Socket was "gracefully closed"';
		wState:=999;
	ELSE (* succesful *)
		sStatus :='Waiting for "OK Packet" from server';
		wState:=70;
	END_CASE

70: (* Wait for "Response" from server *)
	(*diRxCount := SysSockRecv(diSocket 	:= dwSocket,
							 pbyBuffer 	:= ADR(oMySql.abRxBuffer),		(* Address of receive buffer *)
							 diBufferSize:= SIZEOF(oMySql.abRxBuffer),
							 diFlags	:= 0);*)
	diRxCount := SysSockRecv(			hSocket 	:= dwSocket,
										pbyBuffer 	:= ADR(oMySql.abRxBuffer),		(* Address of receive buffer *)
										diBufferSize:= SIZEOF(oMySql.abRxBuffer),
										diFlags		:= 0,
										pResult := ADR(RTS_IEC_RES));
	CASE diRxCount OF
	-1:(* No data available or error occured *)
			; (* Let the watchdog look for *)

	(*0: (* Socket was "gracefully closed"  *)*)
		diError := 16#80001005;
		sStatus :='TCP-ERROR: "SysSockRecv()" returns 0. Socket was "gracefully closed"';
		wState:=999;

	ELSE (* We receive some data from server *)
		IF RTS_IEC_RES <> 0 AND RTS_IEC_RES <> 518 THEN
			diError := 16#80001005;
			sStatus :='TCP-ERROR: "SysSockRecv()" returns 0. Socket was "gracefully closed"';
			wState:=999;
		ELSE
		IF diRxCount > 0 THEN
		dwPacketLength := 	BYTE_TO_DWORD(oMySql.abRxBuffer[0]) OR
							SHL(BYTE_TO_DWORD(oMySql.abRxBuffer[1]),8) OR
							SHL(BYTE_TO_DWORD(oMySql.abRxBuffer[2]),16);
		IF diRxCount >= dwPacketLength THEN
			wState:=75; (* Go ahead *)
		END_IF
		END_IF
		END_IF
	END_CASE

75: (* Check response packet, could be OK- or ERROR-Packet *)
	CASE oMySql.abRxBuffer[4] OF (* field "field_count"*)

	16#00: (* OK-Packet: Identified by "field_count", always = 0 *)
		wState:=90; (* Everything fine - nothing else to do *)

	16#FF: (* ERROR-Packet: Identified by "field_count", always = 16#FF *)
		diError := 16#80005002;
		(* Copy server message into "sStatus"*)
		sStatus :='MYSQL-ERROR:  ';
		pabHelp := ADR(sStatus)+13;
		FOR i:=0 TO DWORD_TO_INT(dwPacketLength-10) DO
			pabHelp^[i] := oMySql.abRxBuffer[13+i];
			IF i>=499 THEN
				EXIT;
			END_IF
		END_FOR
		pabHelp^[i] := 16#00;
		wState:=999;

	ELSE (* Invalid or unexpected response from server (at this time) *)
		diError := 16#80005003;
		sStatus :='MYSQL-ERROR: Invalid or unexpected response from server';
		wState:=999;
	END_CASE

90:	(* Connection established - Free semaphore to allow other function block access to Tx- and Rx-Buffer *)
	SysSemLeave(oMySql.dwBufferSemaphor);
	oMySql.xConnected := TRUE;
	xConnected := oMySql.xConnected;
	IF sDatabase = '' THEN
		sStatus := 'CONNECTED WITH DATABASE';
	ELSE
		sStatus := CONCAT('CONNECTED WITH DATABASE - "', sDatabase);
		sStatus := CONCAT(sStatus, '"');
	END_IF
	xStart := FALSE;
	wState:=100;

100: (* Wait here and check if socket is still alive *)
	IF oMySql.dwSocketHandle = 0 THEN
		xConnected := FALSE;
		sStatus := 'DISCONNECTED';
		wState:=999;
	END_IF
	IF xStart THEN
		wState := 0;
	END_IF

ELSE
	(* Clean up and close connection -----------------------------------------*)
	MySql_Close(oMySql); (* Kill existing connection *)
	xStart := FALSE;
	wState:=0;

END_CASE (**************************************************************************************)

(* Watchdog for statemachine  *)
IF oTON.Q THEN
	xWatchDogOn := FALSE;
	diError := 16#80004001; 	(* Watchdog time elapsed, see sStatus for details *)
	sStatus := CONCAT('TIMEOUT on:', sStatus);
	wState:=999;
END_IF

IF (wState > 0) AND (wState <> 100) THEN
	oTON(IN:=xWatchDogOn , PT:=gcMySql_tTimeOut);
	IF (wStateOld <> wState) THEN
		xWatchDogOn := FALSE; (* Step has changed *)
	ELSE
		xWatchDogOn := TRUE; (* Step still active *)
	END_IF
END_IF
wStateOld:=wState;

END_FUNCTION_BLOCK

// Device/Application/MYSQL/private/MySql_Close
FUNCTION MySql_Close : BOOL
(* This function closes database connection

	Do not "call" this function directly - Use function block "MySql_Logout" 
*)
VAR_IN_OUT
	oMySql : MySql_Context; (* Structure for keeping login and status informations *)
END_VAR
VAR
	i : INT;
END_VAR

IF oMySql.dwSocketHandle <> 0 THEN
	(* Call SysSockShutDown only for IPC's series 758-870  *)
	(*IF ((ADR(%MW0)=16#30000000) OR (ADR(%MW0)=16#20000000)) THEN (* 841 or 88x*)
		;
	ELSE*)
		SysSockShutdown(oMySql.dwSocketHandle, 0);(* 758-870 *)
	(*END_IF*)
	(* Call SysSockClose *)
	SysSockClose( oMySql.dwSocketHandle );
	(* Update context *)
	oMySql.dwSocketHandle := 16#00000000;
	oMySql.xConnected := FALSE;
	(* Clear stServerInfo *)
	oMySql.stServerInfo.bProtocolVersion := 0;
	oMySql.stServerInfo.sServerVersion := '';
	oMySql.stServerInfo.dwThreadId := 0;
	FOR i:=0 TO SIZEOF(oMySql.stServerInfo.abScrambleBuffer) -1 DO
		oMySql.stServerInfo.abScrambleBuffer[i] := 16#00;
	END_FOR
	oMySql.stServerInfo.wServerCapabilities := 16#0000;
	oMySql.stServerInfo.bServerLanguageId := 16#00;
	oMySql.stServerInfo.wServerStatus := 16#00;
	(* Destroy semphore for buffer access synchronization *)
	SysSemDelete(oMySql.dwBufferSemaphor); (* Destroy semaphore  *)
	oMySql.dwBufferSemaphor := 0;
END_IF

END_FUNCTION

// Device/Application/MYSQL/public/MySql_Logout
FUNCTION_BLOCK MySql_Logout
(* This function is used to disconnect from a connected MySQL-Server

	RetVal dwError:	
		16#00000000 => 'SUCCESS'
		16#80001006 => 'TCP-ERROR: "SysSockSend()" returns 0. Socket was "gracefully closed"'
		16#80001007 => 'TCP-ERROR: "SysSockSend()" returns -1'
		16#80004001 => 'TIMEOUT: <actual processed step in state machine>'


 date     | release	| author  | Desc
----------+---------+------------------------------------------------------------
 06.08.10 |  2.0	| CM      | Init 
*)
VAR_INPUT
END_VAR
VAR_IN_OUT
	oMySql : MySql_Context; (* Structure for keeping login and status informations *)
	xStart : BOOL; 			(* Start execution on a rising edge and reset internally when done or on timeout.  *)
END_VAR
VAR_OUTPUT
	diError : DWORD; 		(* Numeric return value - more readable in hex  *)
	sStatus : STRING(200); 	(* Textual description of current state or error *)
END_VAR
VAR
	wState : WORD;	 (* State mashine *)

	oTON			: TON;		(* Watchdogtimer for statemashine *)

	xWatchDogOn		: BOOL; 	(* enable disable Watchdog for statemashine *)
	wStateOld		: WORD;		(* persist the last state of statemashine *)

	xSemaOccupied	: BOOL;		(* This function block instance is current owner of critical path *)

	xResult			: BOOL;		(* Return value of functions *)
	diResult		: __XINT; 	(* Retval value of functions *)

	diTxCount		: __XINT; 	(* Number of bytes to send *)

	(* Helpers *)

	RTS_IEC_RES: UDINT;
END_VAR

CASE  wState OF (* The state maschine *********************************************)

0:	(* Check database connection --------------------------------------------------*)
	IF oMySql.xConnected THEN
		sStatus := 'CONNECTED WITH DATABASE';
		(* Wait for something to do *)
		IF xStart THEN
			diError := 0;
			sStatus := '';
			wState := 5; (* Go ahead *)
		END_IF
	ELSE
		IF xStart THEN
			xStart := FALSE;
		END_IF
		sStatus :='DISCONNECTED';
	END_IF

5: (* Wait until semaphore for Rx- and Tx-Buffer synchronization is available.
	With SysSemTry (which always returns immediately), a semaphore will be marked as used. 
	The returnvalue is TRUE if this succeeded and FALSE if the semaphore is already used by another task.  *)
	sStatus := 'Wait for semaphor';
	
	RTS_IEC_RES := SysSemTry(oMySql.dwBufferSemaphor);
	xResult := (RTS_IEC_RES = 0);
	IF xResult THEN
		xSemaOccupied := TRUE;
		sStatus := 'Close Database connection';
		wState:=10; (* Go ahead *)
	END_IF

10: (*Prepare command packet "COM_QUIT"  ----------------------------------------*)
	(* Packet-Length - will be calculated and assigned at the end of this step *)
	oMySql.abTxBuffer[ 0] := 16#01;
	oMySql.abTxBuffer[ 1] := 16#00;
	oMySql.abTxBuffer[ 2] := 16#00;
	(* Packet-Number *)
	oMySql.abTxBuffer[ 3] := 0;
	(* Command-Type *)
	oMySql.abTxBuffer[ 4] := 16#01;  (* COM_QUIT - mysql_close *)
	(* No additional Command-Argument *)
	diTxCount := 5; (* Bytes to send *)
	wState:=20; (* Go ahead *)

20: (* Send command packet "COM_QUERY"  ---------------------------*)
	diResult := SysSockSend(	hSocket := oMySql.dwSocketHandle,
								pbyBuffer := ADR(oMySql.abTxBuffer),
								diBufferSize := diTxCount,
								diFlags := 0,
								pResult := ADR(RTS_IEC_RES));

	CASE diResult OF
	-1:	(* ERROR *)
		diError := 16#80001007;
		sStatus :='TCP-ERROR: "SysSockSend()" returns -1';
	0: (* Socket was "gracefully closed" *)
		diError := 16#80001006;
		sStatus :='TCP-ERROR: "SysSockSend()" returns 0. Socket was "gracefully closed"';
	ELSE (* succesful *)
		(* Server will close TCP-Connection immidiadly *)
		;
	END_CASE
	wState:=999;

ELSE
	(* Clean up and destroy semaphore -----------------------------------------*)
	IF xSemaOccupied THEN
		xSemaOccupied := FALSE;
		SysSemLeave(oMySql.dwBufferSemaphor); (* Leave semaphore, to be shure nowbody is blocked by her *)
	END_IF
	MySql_Close(oMySql); (* Kill existing connection *)
	sStatus := 'DISCONNECTED';
	xStart := FALSE;
	wState:=0;

END_CASE (**************************************************************************************)

(* Watchdog for statemachine  *)
IF oTON.Q THEN
	xWatchDogOn := FALSE;
	diError := 16#80004001; 	(* Watchdog time elapsed, see sStatus for details *)
	sStatus := CONCAT('TIMEOUT on:', sStatus);
	wState:=999;
END_IF

IF (wState > 0) THEN
	oTON(IN:=xWatchDogOn , PT:=gcMySql_tTimeOut);
	IF (wStateOld <> wState) THEN
		xWatchDogOn := FALSE; (* Step has changed *)
	ELSE
		xWatchDogOn := TRUE; (* Step still active *)
	END_IF
END_IF
wStateOld:=wState;

END_FUNCTION_BLOCK

// Device/Application/MYSQL/private/MySql_Scramble
FUNCTION MySql_Scramble : BOOL
(* 	This function is used by client to create authenticated reply to the
   	server's greeting.
	Produce an obscure octet sequence from password and random
	string, recieved from the server. This sequence corresponds to the
	password, but password can not be easily restored from it. The sequence
	then sent to the server for validation. Trailing zero is not stored
	in the buf as it is not needed.

	Returns: TRUE if successful, FALSE if it failed. 
*)
VAR CONSTANT
	SHA1_HASH_SIZE : UINT := 20;
END_VAR
VAR_INPUT
	abMessage: ARRAY [0..SHA1_HASH_SIZE] OF BYTE; (*   IN  random message, must be exactly SCRAMBLE_LENGTH long and NULL-terminated. *)
	sPassword: STRING; (*  IN  users' password *)
END_VAR
VAR_IN_OUT
	abScrambleBuffer : ARRAY [0..SHA1_HASH_SIZE] OF BYTE; (* OUT store scrambled string here. The buf must be at least SHA1_HASH_SIZE bytes long. *)
END_VAR
VAR
	sha : SHA1Context ;   						(* SHA-1 context   *)
	abHashStage1 : ARRAY [0..SHA1_HASH_SIZE] OF BYTE;
	abHashStage2 : ARRAY [0..SHA1_HASH_SIZE] OF BYTE;

	i : INT;
	pabHelp : POINTER TO ARRAY [0..40] OF BYTE;
END_VAR

(* Reset the SHA-1 context and process input *)
SHA1Reset(ADR(sha));
(* stage 1: hash password *)
SHA1Input(ADR(sha), ADR(sPassword), LEN(sPassword));
IF NOT SHA1Result(ADR(sha), abHashStage1) THEN
	(* On Error *)
	MySql_Scramble := FALSE;
	RETURN;
END_IF
(* stage 2: hash stage 1; note that hash_stage2 is stored in the database *)
SHA1Reset(ADR(sha));
SHA1Input(ADR(sha), ADR(abHashStage1), SHA1_HASH_SIZE);
IF NOT SHA1Result(ADR(sha), abHashStage2) THEN
	(* On Error *)
	MySql_Scramble := FALSE;
	RETURN;
END_IF
(* Create crypt string as sha1(message, hash_stage2) *)
SHA1Reset(ADR(sha));
SHA1Input(ADR(sha), ADR(abMessage), SHA1_HASH_SIZE);
SHA1Input(ADR(sha), ADR(abHashStage2), SHA1_HASH_SIZE);
(* XOR allows 'from' and 'to' overlap: lets take advantage of it *)
IF NOT SHA1Result(ADR(sha), abScrambleBuffer) THEN
	(* On Error *)
	MySql_Scramble := FALSE;
	RETURN;
END_IF
(* Simple XOR is used here but it is OK as we crypt random strings.
Note, that XOR(s1, XOR(s1, s2)) == s2, XOR(s1, s2) == XOR(s2, s1) *)
pabHelp := ADR(abHashStage1);
FOR i:=0 TO SHA1_HASH_SIZE -1 DO
	abScrambleBuffer[i] := abScrambleBuffer[i] XOR pabHelp^[i];
END_FOR
MySql_Scramble := TRUE;


(*
00434   sha1_reset(&sha1_context);
00435   /* stage 1: hash password */
00436   sha1_input(&sha1_context, password, (uint) strlen(password));
00437   sha1_result(&sha1_context, hash_stage1);
00438   /* stage 2: hash stage 1; note that hash_stage2 is stored in the database */
00439   sha1_reset(&sha1_context);
00440   sha1_input(&sha1_context, hash_stage1, SHA1_HASH_SIZE);
00441   sha1_result(&sha1_context, hash_stage2);
00442   /* create crypt string as sha1(message, hash_stage2) */;
00443   sha1_reset(&sha1_context);
00444   sha1_input(&sha1_context, message, SCRAMBLE_LENGTH);
00445   sha1_input(&sha1_context, hash_stage2, SHA1_HASH_SIZE);
00446   /* xor allows 'from' and 'to' overlap: lets take advantage of it */
00447   sha1_result(&sha1_context,  to);
00448   my_crypt(to, to, hash_stage1, SCRAMBLE_LENGTH);
00449 }
00450
*)

(*
###############################################################################
0357     Encrypt/Decrypt function used for password encryption in authentication.
00358     Simple XOR is used here but it is OK as we crypt random strings. Note,
00359     that XOR(s1, XOR(s1, s2)) == s2, XOR(s1, s2) == XOR(s2, s1)
00360   SYNOPSIS
00361     my_crypt()
00362     to      OUT buffer to hold crypted string; must be at least len bytes
00363                 long; to and s1 (or s2) may be the same.
00364     s1, s2  IN  input strings (of equal length)
00365     len     IN  length of s1 and s2
00366 */
00367 
00368 static void
00369 my_crypt(char *to, const uchar *s1, const uchar *s2, uint len)
00370 {
00371   const uint8 *s1_end= s1 + len;
00372   while (s1 < s1_end)
00373     *to++= *s1++ ^ *s2++;
00374 }

*)

END_FUNCTION

// Device/Application/MYSQL/private/SHA/SHA1Reset
FUNCTION SHA1Reset : BOOL
(* This function will initialize the SHA1Context in preparation for computing a new message digest *)
VAR_INPUT
	context : POINTER TO SHA1Context;
END_VAR
VAR
END_VAR

context^.Length_Low             := 0;
context^.Length_High            := 0;
context^.Message_Block_Index    := 0;
context^.Message_Digest[0]      := 16#67452301;
context^.Message_Digest[1]      := 16#EFCDAB89;
context^.Message_Digest[2]      := 16#98BADCFE;
context^.Message_Digest[3]      := 16#10325476;
context^.Message_Digest[4]      := 16#C3D2E1F0;
context^.Computed   := FALSE;
context^.Corrupted  := FALSE;

END_FUNCTION

// Device/Application/MYSQL/private/SHA/SHA1Input
FUNCTION SHA1Input : BOOL
(* This function accepts an array of octets as the next portion of
   the message*)
VAR_INPUT
	context : POINTER TO SHA1Context; (* The SHA-1 context to update *)
	message_array: POINTER TO BYTE;  (* An array of characters representing the next portion of the message.*)
	length: UINT;          			  (* The length of the message in message_array *)
END_VAR
VAR
END_VAR

IF (length <= 0)THEN
	RETURN;
END_IF

IF (context^.Computed OR context^.Corrupted) THEN
	context^.Corrupted := 1;
	RETURN;
END_IF

WHILE( length>0 AND (NOT context^.Corrupted) )DO
	context^.Message_Block[context^.Message_Block_Index] := (message_array^ AND 16#FF);
	context^.Message_Block_Index := context^.Message_Block_Index +1;
	context^.Length_Low := context^.Length_Low +8;
    (* Force it TO 32 bits *)
	context^.Length_Low := context^.Length_Low AND 16#FFFFFFFF;
    IF (context^.Length_Low = 0) THEN
		context^.Length_High := context^.Length_High +1;
		(* Force it TO 32 bits *)
		context^.Length_High := context^.Length_High AND 16#FFFFFFFF;
		IF (context^.Length_High = 0) THEN
			(* Message is too long *)
			context^.Corrupted := 1;
		END_IF
	END_IF

	IF (context^.Message_Block_Index = 64) THEN
		SHA1ProcessMessageBlock(context);
	END_IF

	message_array := message_array +1;
	length := length -1;
END_WHILE

END_FUNCTION

// Device/Application/MYSQL/private/SHA/SHA1ProcessMessageBlock
FUNCTION SHA1ProcessMessageBlock : BOOL
(* 	This function will process the next 512 bits of the message
	stored in the Message_Block array.

	Many of the variable names in the SHAContext, especially the
	single character names, were used because those were the names
	used in the publication.
*)
VAR_INPUT
	context : POINTER TO SHA1Context;
END_VAR
VAR CONSTANT
	K : ARRAY [0..3] OF DWORD := [16#5A827999, 16#6ED9EBA1, 16#8F1BBCDC, 16#CA62C1D6];
	
END_VAR
VAR
	t : INT; (* Loop counter *)
	temp : DWORD; (* Temporary word value*)
	W : ARRAY [0..79] OF DWORD; (* Word sequence*)
	A, B, C, D, E : DWORD; (* Word buffers *)

END_VAR

(*  Define the circular shift macro
#define SHA1CircularShift(bits,word) 
	((((word) << (bits)) & 0xFFFFFFFF) | ((word) >> (32-(bits))))

	(SHL(word, bits) AND 16#FFFFFFFF) OR SHR(word,(32-bits));
*)

(* Initialize the first 16 dwords in the array W *)

FOR t:=0 TO 15 DO
	W[t] := 		SHL(BYTE_TO_DWORD(context^.Message_Block[(t * 4)+ 0]), 24);
	W[t] := W[t] OR SHL(BYTE_TO_DWORD(context^.Message_Block[(t * 4)+ 1]), 16);
	W[t] := W[t] OR SHL(BYTE_TO_DWORD(context^.Message_Block[(t * 4)+ 2]),  8);
	W[t] := W[t] OR    (BYTE_TO_DWORD(context^.Message_Block[(t * 4)+ 3])    );
END_FOR

FOR t:=16 TO 79 DO
	temp := W[t-3] XOR W[t-8] XOR W[t-14] XOR W[t-16];
	(* W[t] := SHA1CircularShift(1, temp); *)
	W[t] := (SHL(temp, 1) AND 16#FFFFFFFF) OR SHR(temp,(32-1));
END_FOR

A := context^.Message_Digest[0];
B := context^.Message_Digest[1];
C := context^.Message_Digest[2];
D := context^.Message_Digest[3];
E := context^.Message_Digest[4];

FOR t:=0 TO 19 DO
	(*temp := SHA1CircularShift(5,A);*)
	temp := (SHL(A, 5) AND 16#FFFFFFFF) OR SHR(A,(32-5));
	temp := temp + ((B AND C) OR (NOT(B) AND D)) + E + W[t] + K[0];
	temp := temp AND 16#FFFFFFFF;
	E := D;
	D := C;
	(*C := SHA1CircularShift(30,B);*)
	C := (SHL(B, 30) AND 16#FFFFFFFF) OR SHR(B,(32-30));
	B := A;
	A := temp;
END_FOR

FOR t:=20 TO 39 DO
	(*temp := SHA1CircularShift(5,A);*)
	temp := (SHL(A, 5) AND 16#FFFFFFFF) OR SHR(A,(32-5));
	temp := temp + (B XOR C XOR D) + E + W[t] + K[1];
	temp := temp AND 16#FFFFFFFF;
	E := D;
	D := C;
	(*C := SHA1CircularShift(30,B);*)
	C := (SHL(B, 30) AND 16#FFFFFFFF) OR SHR(B,(32-30));
	B := A;
	A := temp;
END_FOR

FOR t:=40 TO 59 DO
	(*temp := SHA1CircularShift(5,A);*)
	temp := (SHL(A, 5) AND 16#FFFFFFFF) OR SHR(A,(32-5));
	temp := temp + ((B AND C) OR (B AND D) OR (C AND D)) + E + W[t] + K[2];
	temp := temp AND 16#FFFFFFFF;
	E := D;
	D := C;
	(*C := SHA1CircularShift(30,B);*)
	C := (SHL(B, 30) AND 16#FFFFFFFF) OR SHR(B,(32-30));
	B := A;
	A := temp;
END_FOR

FOR t:=60 TO 79 DO
	(*temp := SHA1CircularShift(5,A);*)
	temp := (SHL(A, 5) AND 16#FFFFFFFF) OR SHR(A,(32-5));
	temp := temp + (B XOR C XOR D) + E + W[t] + K[3];
	temp := temp AND 16#FFFFFFFF;
	E := D;
	D := C;
	(*C := SHA1CircularShift(30,B);*)
	C := (SHL(B, 30) AND 16#FFFFFFFF) OR SHR(B,(32-30));
	B := A;
	A := temp;
END_FOR



context^.Message_Digest[0] := (context^.Message_Digest[0] + A) AND 16#FFFFFFFF;
context^.Message_Digest[1] := (context^.Message_Digest[1] + B) AND 16#FFFFFFFF;
context^.Message_Digest[2] := (context^.Message_Digest[2] + C) AND 16#FFFFFFFF;
context^.Message_Digest[3] := (context^.Message_Digest[3] + D) AND 16#FFFFFFFF;
context^.Message_Digest[4] := (context^.Message_Digest[4] + E) AND 16#FFFFFFFF;

context^.Message_Block_Index := 0;

END_FUNCTION

// Device/Application/MYSQL/private/SHA/SHA1Result
FUNCTION SHA1Result : BOOL
(* This function will return the 160-bit message digest into the Message_Digest array within the SHA1Context provided
	
	Returns: TRUE if successful, FALSE if it failed. 
*)
VAR_INPUT
	context : POINTER TO SHA1Context;
END_VAR
VAR_IN_OUT
	abDigest : ARRAY [0..20] OF BYTE;
END_VAR
VAR
	adwDigest : ARRAY [0..4] OF DWORD;
	i, j : INT;
	dwMaskByte : DWORD := 16#000000FF;
END_VAR

IF (context^.Corrupted) THEN
	SHA1Result := FALSE;
	RETURN;
END_IF

IF (NOT context^.Computed) THEN
	SHA1PadMessage(context);
    context^.Computed := TRUE;
END_IF

(* Copy Digest to output *)
FOR i:=0 TO 4 DO
	adwDigest[i] := context^.Message_Digest[i];
	(* Convert Digest to ArrayOfByte *)
	FOR j:=0 TO 3 DO
		abDigest[(i*4)+j]:= DWORD_TO_BYTE(SHR(adwDigest[i], 24-(j*8)) AND dwMaskByte);
	END_FOR
END_FOR


SHA1Result := TRUE;

END_FUNCTION

// Device/Application/MYSQL/private/SHA/SHA1PadMessage
FUNCTION SHA1PadMessage : BOOL
(* 	According to the standard, the message must be padded to an even
   	512 bits.  The first padding bit must be a '1'.  The last 64
	bits represent the length of the original message.  All bits in
	between should be 0.  This function will pad the message
	according to those rules by filling the Message_Block array
	accordingly.  It will also call SHA1ProcessMessageBlock()
	appropriately.  When it returns, it can be assumed that the
	message digest has been computed.*)
VAR_INPUT
	context : POINTER TO SHA1Context;
END_VAR
VAR
END_VAR

(* 	Check to see if the current message block is too small to hold
	the initial padding bits and length.  If so, we will pad the
	block, process it, and then continue padding into a second
	block.*)

IF (context^.Message_Block_Index > 55) THEN
	context^.Message_Block[context^.Message_Block_Index] := 16#80;
	context^.Message_Block_Index := context^.Message_Block_Index +1;
    WHILE(context^.Message_Block_Index < 64) DO
    	context^.Message_Block[context^.Message_Block_Index] := 0;
		context^.Message_Block_Index := context^.Message_Block_Index +1;
    END_WHILE

	SHA1ProcessMessageBlock(context);

    WHILE(context^.Message_Block_Index < 56) DO
		context^.Message_Block[context^.Message_Block_Index] := 0;
		context^.Message_Block_Index := context^.Message_Block_Index +1;
	END_WHILE
ELSE

	context^.Message_Block[context^.Message_Block_Index] := 16#80;
	context^.Message_Block_Index := context^.Message_Block_Index +1;
    WHILE(context^.Message_Block_Index < 56) DO
		context^.Message_Block[context^.Message_Block_Index] := 0;
		context^.Message_Block_Index := context^.Message_Block_Index +1;
    END_WHILE
END_IF

(* Store the message length as the last 8 octets *)
context^.Message_Block[56] := DWORD_TO_BYTE(SHR(context^.Length_High, 24) AND 16#000000FF);
context^.Message_Block[57] := DWORD_TO_BYTE(SHR(context^.Length_High,16) AND 16#000000FF);
context^.Message_Block[58] := DWORD_TO_BYTE(SHR(context^.Length_High, 8) AND 16#000000FF);
context^.Message_Block[59] := DWORD_TO_BYTE((context^.Length_High) AND 16#000000FF);
context^.Message_Block[60] := DWORD_TO_BYTE(SHR(context^.Length_Low, 24) AND 16#000000FF);
context^.Message_Block[61] := DWORD_TO_BYTE(SHR(context^.Length_Low, 16) AND 16#000000FF);
context^.Message_Block[62] := DWORD_TO_BYTE(SHR(context^.Length_Low, 8) AND 16#000000FF);
context^.Message_Block[63] := DWORD_TO_BYTE((context^.Length_Low) AND 16#000000FF);

SHA1ProcessMessageBlock(context);

END_FUNCTION

// Device/Application/MYSQL/private/SHA/SHA1
FUNCTION SHA1 : BOOL
(* This function provide the Secure Hashing Standard as defined
   in FIPS PUB 180-1 published April 17, 1995.
*)
VAR_INPUT
	pbMessage : POINTER TO BYTE; (* Start address of message to hash *)
	iByteCount : INT; 			(* Number of bytes to hash or message length *)
END_VAR
VAR_IN_OUT
	abDigest : ARRAY [0..20] OF BYTE;
	sDigest : STRING(80);
END_VAR
VAR
	sha : SHA1Context ;   (* SHA-1 context                 *)
	adwDigest : ARRAY [0..4] OF DWORD;
	i, k, j : INT;
	pabHelp : POINTER TO ARRAY [0..40] OF BYTE;
	bHelp : BYTE;
	dwMaskByte : DWORD := 16#000000FF;
	dwMaskNibble : DWORD := 16#0000000F;



END_VAR

(* Reset the SHA-1 context and process input *)
SHA1Reset(ADR(sha));

SHA1Input(ADR(sha), pbMessage, iByteCount);

IF SHA1Result(ADR(sha), abDigest) THEN

	sDigest := SHA1Hex2String(abDigest);

	SHA1 := TRUE;
ELSE
	SHA1 := FALSE;
END_IF

END_FUNCTION

// Device/Application/MYSQL/private/SHA/SHA1Hex2String
FUNCTION SHA1Hex2String : STRING
(* This function convert the binary digest into a readable string *)
VAR_INPUT
	abDigest : ARRAY [0..20] OF BYTE;
END_VAR
VAR
	bHelp : BYTE;
	abHelp : ARRAY [0..40] OF BYTE;
	bMaskNibble : BYTE := 16#0F;
	psHelp : POINTER TO STRING;
	i : INT;
END_VAR

(* Convert Digest to STRING *)
FOR i:=0 TO 19 DO
	(* Convert upper nibble *)
	bHelp := SHR(abDigest[i], 4) AND bMaskNibble;
	IF bHelp <= 9 THEN
		abHelp[i*2]:= bHelp + 16#30;
	ELSE
		abHelp[i*2]:= 55 + bHelp;
	END_IF
	(* Convert upper nibble *)
	bHelp := abDigest[i] AND bMaskNibble;
	IF bHelp <= 9 THEN
		abHelp[(i*2)+1]:= bHelp + 16#30;
	ELSE
		abHelp[(i*2)+1]:= 55 + bHelp;
	END_IF
END_FOR
abHelp[40] := 16#00;
psHelp := ADR(abHelp);
SHA1Hex2String := psHelp^;

END_FUNCTION

// Device/Application/MYSQL/public/MySql_Execute
FUNCTION_BLOCK MySql_Execute
(* This function block is used to send SQL statements to server who
   do not respond with result sets, such as:
		INSERT, UPDATE, DELETE, ALTER, DROP, ...

	RetVal dwError:	
		16#00000000 => 'SUCCESS'
		16#80001005 => 'TCP-ERROR: "SysSockRecv()" returns 0. Socket was "gracefully closed"'
		16#80001006 => 'TCP-ERROR: "SysSockSend()" returns 0. Socket was "gracefully closed"'
		16#80001007 => 'TCP-ERROR: "SysSockSend()" returns -1'
		16#80005002 => 'MYSQL-ERROR: <Message from server>	
		16#80005003 => 'MYSQL-ERROR: Invalid or unexpected response from server'
		16#80005005 => 'MYSQL-ERROR: Not connected with database, LOGIN before use'
		16#80004001 => 'TIMEOUT: <actual processed step in state machine>'


	Remarks for "asSqlStatement":
	You can modify the "length" and number of elements in "asSqlStatement" by hiding 
	libraries global constants with global constants of same name in your project:
		- gcMySql_iSqlUpperBound:
				Defines the UpperBound of "asSqlStatement", to provide an SQL statement 
				as "ARRAY [0..UpperBound] OF STRING(Size)" 
		- gcMySql_iSqlLength:
				Defines the Size in byte of an array element of "asSqlStatement", 
				to provide an SQL statement as "ARRAY [0..UpperBound] OF STRING(Size)".   

	All non numeric SQL param values must be "quoted" with an apostroph(').
	Apostroph(') is also CoDesys-String-Start-End-Identifier.
	To use an apostroph(') inside a CoDeSys-String type $27 or $'.

	Example: 
		(* Prepare SQL-Insert-Statement *)	
		asSqlStatement1[0] := 'INSERT INTO atable ';	
		asSqlStatement1[1] := '( aBool, aByte, aWord, aDint, aReal, ';	
		asSqlStatement1[2] := '  aString, aDT, aTime, aUdint ) ';	
		asSqlStatement1[3] := 'VALUES ';	
		asSqlStatement1[4] := '( TRUE, 17, 32333, 1111111, 1.42, ';	
		asSqlStatement1[5] := ' $'Hallo$', $'2010-08-13 11:56:42$', ';	
		asSqlStatement1[6] := ' $'13:12:57$', 62222 )';	
		asSqlStatement1[7] := ''; (* End of SQL-Statement *)

	Restriction: 
		- Maximum length for identifiers are 250 bytes!


 date     | release	| author  | Desc
----------+---------+------------------------------------------------------------
 25.01.12 |  3.4	| CM      | Bugfix for transmit large SQL statements 
 24.01.12 |  3.4	| CM      | Bugfix for christmas tree on large error response 
 06.08.10 |  2.0	| CM      | Init 
 
*)
VAR_INPUT
	asSqlCommand : ARRAY [0..gcMySql_iSqlUpperBound] OF STRING(gcMySql_iSqlLength);
END_VAR
VAR_IN_OUT
	oMySql : MySql_Context; (* Structure for keeping login and status informations *)
	xStart : BOOL; 			(* Start execution on a rising edge and reseted internally when done or on timeout.  *)
END_VAR
VAR_OUTPUT
	diError : DWORD; 		(* Numeric return value - more readable in hex  *)
	sStatus : STRING(200); 	(* Textual description of current state or error *)
END_VAR
VAR
	wState : WORD;	 (* State mashine *)

	oTON			: TON;	(* Watchdogtimer for statemashine *)

	xWatchDogOn		: BOOL; (* enable disable Watchdog for statemashine *)
	wStateOld		: WORD;	(* persist the last state of statemashine *)

	xSemaOccupied	: BOOL;	(* This function block instance is current owner of critical path *)

	xResult			: BOOL;	(* Return value of functions *)
	diResult		: __XINT; (* Retval value of functions *)

	diTxCount		: __XINT; (* Number of bytes to send *)
	pbTxBufferPos	: POINTER TO BYTE; (* Position in Tx buffer of next data to transmit *)
	oTonTxDelay 	: TON; (* Delay for transmitting the rest package *)
	diRxCount		: __XINT; (* Number of received bytes *)

	(* Helpers *)
	dwPacketLength : DWORD; (*  *)
	uiPos : UINT;

	dwMask : DWORD := 16#000000FF;

	i, k : INT;
	dwHelp : DWORD;
	iHelp : INT;
	pabHelp : POINTER TO ARRAY [0..512] OF BYTE;
	RTS_IEC_RES: UDINT;
	ptrDINT : POINTER TO DINT;
END_VAR

CASE  wState OF (* The state maschine *********************************************)

0:	(* Idle - wait for something to do -------------------------------------------*)
	IF xStart THEN
		diError := 0;
		wState:=5; (* Go ahead *)
	END_IF

5: (* Check database connection --------------------------------------------------*)
	IF oMySql.xConnected THEN
		wState:=10; (* Go ahead *)
	ELSE
		diError := 16#80005005;
		sStatus :='MYSQL-ERROR: Not connected with database, LOGIN before use';
		wState:=999;
	END_IF

10: (* Wait until semaphore for Rx- and Tx-Buffer synchronization is available.
	With SysSemTry (which always returns immediately), a semaphore will be marked as used. 
	The returnvalue is TRUE if this succeeded and FALSE if the semaphore is already used by another task.  *)
	sStatus := 'Wait for semaphor';
	RTS_IEC_RES := SysSemTry(oMySql.dwBufferSemaphor);
	xResult := (RTS_IEC_RES = 0);
	IF xResult THEN
		xSemaOccupied := TRUE;
		sStatus := 'Execute SQL command';
		wState:=20; (* Go ahead *)
	END_IF

20: (*Prepare command packet "COM_QUERY"  ----------------------------------------*)
	(* Packet-Length - will be calculated and assigned at the end of this step *)
	oMySql.abTxBuffer[ 0] := 16#00;
	oMySql.abTxBuffer[ 1] := 16#00;
	oMySql.abTxBuffer[ 2] := 16#00;
	(* Packet-Number *)
	oMySql.abTxBuffer[ 3] := 0;
	(* Command-Type *)
	oMySql.abTxBuffer[ 4] := 16#03;  (* COM_QUERY - mysql_real_query *)
	(* Command-Argument (Null-Terminated String)*)
	uiPos := 5;
	FOR k:=0 TO gcMySql_iSqlUpperBound DO
		IF asSqlCommand[k] <> '' THEN
			pabHelp := ADR(asSqlCommand[k]);
			iHelp := LEN(asSqlCommand[k]);
			FOR i:=0 TO iHelp-1 DO
				oMySql.abTxBuffer[uiPos+i] := pabHelp^[i];
			END_FOR
			uiPos := uiPos + iHelp;
		ELSE
			EXIT;
		END_IF
	END_FOR
	oMySql.abTxBuffer[uiPos] := 16#00; (* Append STRING_END character "/0" *)
	uiPos := uiPos +1;

	(* Calculate number of bytes to transmit and logical packet-length *)
	diTxCount := uiPos; (* Bytes to send *)
	dwPacketLength := uiPos -4;
	(* Packet-Length *)
	oMySql.abTxBuffer[ 0] := DWORD_TO_BYTE(dwPacketLength AND dwMask);
	oMySql.abTxBuffer[ 1] := DWORD_TO_BYTE(SHR(dwPacketLength, 8) AND dwMask);
	oMySql.abTxBuffer[ 2] := DWORD_TO_BYTE(SHR(dwPacketLength, 16) AND dwMask);
	(* Set TxBufferPointer to begin of abTxBuffer *)
	pbTxBufferPos := ADR(oMySql.abTxBuffer);
	wState:=25; (* Go ahead *)

25: (* Send command packet "COM_QUERY"  ---------------------------*)
	(*diResult := SysSockSend(diSocket := oMySql.dwSocketHandle,
							pbyBuffer := pbTxBufferPos,
							diBufferSize := diTxCount,
							diFlags := 0);*)
	diResult := SysSockSend(		hSocket := oMySql.dwSocketHandle,
								  	pbyBuffer := pbTxBufferPos,
								  	diBufferSize := diTxCount,
								  	diFlags := 0,
									pResult := ADR(RTS_IEC_RES));
									

	CASE diResult OF
	-1:	(* ERROR *)
		diError := 16#80001007;
		sStatus :='TCP-ERROR: "SysSockSend()" returns -1';
		wState:=999;
	0: (* Socket was "gracefully closed" *)
		diError := 16#80001006;
		sStatus :='TCP-ERROR: "SysSockSend()" returns 0. Socket was "gracefully closed"';
		wState:=999;
	ELSE (* succesful *)
		IF diResult >= diTxCount THEN
			(* All data transmitted *)
			wState:=30;
		ELSE
			(* Wait 200ms and then try to send the rest *)
			diTxCount := diTxCount - diResult;
			ptrDINT := ADR(diResult);
			pbTxBufferPos := pbTxBufferPos + ptrDINT^;
			wState:=27;
		END_IF
	END_CASE

27: (* Wait max ACK time (200ms) before send the rest, to support very slow servers also.
	   Function SysSockSend() will return -1 (Window Full) when you try to send the next 
	   package, before the last package are "ACKnoledged" by peer. *)
	oTonTxDelay(IN:=TRUE , PT:= t#200ms );
	IF oTonTxDelay.Q THEN
		oTonTxDelay(IN:=FALSE);
		wState := 25;
	END_IF

30: (* Wait for "Response" packet *)
	(*diRxCount := SysSockRecv(diSocket 	:= oMySql.dwSocketHandle,
							 pbyBuffer 	:= ADR(oMySql.abRxBuffer),		(* Address of receive buffer *)
							 diBufferSize:= SIZEOF(oMySql.abRxBuffer),
							 diFlags	:= 0);*)
	diRxCount := SysSockRecv(			hSocket 	:= oMySql.dwSocketHandle,
										pbyBuffer 	:= ADR(oMySql.abRxBuffer),		(* Address of receive buffer *)
										diBufferSize:= SIZEOF(oMySql.abRxBuffer),
										diFlags		:= 0,
										pResult := ADR(RTS_IEC_RES));
	CASE diRxCount OF
	-1:(* No data available or error occured *)
			; (* Let the watchdog look for *)

	(*0: (* Socket was "gracefully closed"  *)*)
		MySql_Close(oMySql);
		diError := 16#80001005;
		sStatus :='TCP-ERROR: "SysSockRecv()" returns 0. Socket was "gracefully closed"';
		wState:=999;

	ELSE (* We receive some data from server *)
		IF RTS_IEC_RES <> 0 AND RTS_IEC_RES <> 518 THEN
			diError := 16#80001005;
			sStatus :='TCP-ERROR: "SysSockRecv()" returns 0. Socket was "gracefully closed"';
			wState:=999;
		ELSE
		dwPacketLength := 	BYTE_TO_DWORD(oMySql.abRxBuffer[0]) OR
							SHL(BYTE_TO_DWORD(oMySql.abRxBuffer[1]),8) OR
							SHL(BYTE_TO_DWORD(oMySql.abRxBuffer[2]),16);
		IF diRxCount >= dwPacketLength THEN
			wState:=35; (* Go ahead *)
		END_IF
		END_IF
	END_CASE

35: (* Check response packet, could be OK- or ERROR-Packet *)
	CASE oMySql.abRxBuffer[4] OF (* field "field_count"*)
	16#00: (* OK-Packet: Identified by "field_count", always = 0 *)
		(* Read "effected rows" - (length coded binary*)
		CASE oMySql.abRxBuffer[5] OF
		252: (* Value of "effected rows" are stored in following 16-bit (2 bytes) *)
			dwHelp := 	BYTE_TO_DWORD(oMySql.abRxBuffer[6]) 	OR
					SHL(BYTE_TO_DWORD(oMySql.abRxBuffer[7]),8);
			sStatus := CONCAT('Successful executed - affected rows: ', DWORD_TO_STRING(dwHelp));

		253: (* Value of "effected rows" are stored in following 24-bit (3 bytes) *)
			dwHelp := 	BYTE_TO_DWORD(oMySql.abRxBuffer[6]) 	OR
					SHL(BYTE_TO_DWORD(oMySql.abRxBuffer[7]),8) 	OR
					SHL(BYTE_TO_DWORD(oMySql.abRxBuffer[8]),16);
			sStatus := CONCAT('Successful executed - affected rows: ', DWORD_TO_STRING(dwHelp));

		254: (* Value of "effected rows" are stored in following 64-bit (8 bytes) *)
			sStatus := 'Successful executed - affected rows: "very very mutch"';

		ELSE
			(* Value of "effected rows" himselve *)
			sStatus := CONCAT('Successful executed - affected rows: ', BYTE_TO_STRING(oMySql.abRxBuffer[5]));
		END_CASE
		wState:=999;

	16#FF: (* ERROR-Packet: Identified by "field_count", always = 16#FF *)
		diError := 16#80005002;
		(* Copy server message into "sStatus"*)
		sStatus :='MYSQL-ERROR:  ';
		pabHelp := ADR(sStatus)+13;
		FOR i:=0 TO DWORD_TO_INT(dwPacketLength -10) DO
			pabHelp^[i] := oMySql.abRxBuffer[13+i];
			IF i>=180 THEN
				EXIT;
			END_IF
		END_FOR
		pabHelp^[i] := 16#00;
		wState:=999;

	ELSE (* Invalid or unexpected response from server (at this time) *)
		diError := 16#80005003;
		sStatus :='MYSQL-ERROR: Invalid or unexpected response from server';
		wState:=999;
	END_CASE

ELSE
	(* Clean up and leave connection open -----------------------------------------*)
	IF xSemaOccupied THEN
		SysSemLeave(oMySql.dwBufferSemaphor); (* Leave semaphore, to be shure nowbody is blocked by her *)
		xSemaOccupied := FALSE;
	END_IF
	xStart := FALSE;
	wState:=0;

END_CASE (**************************************************************************************)

(* Watchdog for statemachine  *)
IF oTON.Q THEN
	xWatchDogOn := FALSE;
	diError := 16#80004001; 	(* Watchdog time elapsed, see sStatus for details *)
	sStatus := CONCAT('TIMEOUT on:', sStatus);
	wState:=999;
END_IF

IF (wState > 0) THEN
	oTON(IN:=xWatchDogOn , PT:=gcMySql_tTimeOut);
	IF (wStateOld <> wState) THEN
		xWatchDogOn := FALSE; (* Step has changed *)
	ELSE
		xWatchDogOn := TRUE; (* Step still active *)
	END_IF
END_IF
wStateOld:=wState;

END_FUNCTION_BLOCK

// Device/Application/MYSQL/public/MySql_Query
FUNCTION_BLOCK MySql_Query
(* This function block is used to send SQL "SELECT" statements to server who
   respond with result sets.

	RetVal dwError:	
		16#00000000 => 'SUCCESS'
		16#80001005 => 'TCP-ERROR: "SysSockRecv()" returns 0. Socket was "gracefully closed"'
		16#80001006 => 'TCP-ERROR: "SysSockSend()" returns 0. Socket was "gracefully closed"'
		16#80001007 => 'TCP-ERROR: "SysSockSend()" returns -1'
		16#80001008 => 'TCP-ERROR: Receive buffer to small - increase '
		16#80005002 => 'MYSQL-ERROR: <Message from server>	
		16#80005003 => 'MYSQL-ERROR: Invalid or unexpected response from server'
		16#80005005 => 'MYSQL-ERROR: Not connected with database, LOGIN before use'
		16#80005006 => 'MYSQL-ERROR: Result set has more columns then defined in "gcMySql_dwMaxColumnCount" '
		16#80005007 => 'MYSQL-ERROR: Unsupported value for "column count", provided as 64-bit value(8 bytes) in "Result-Set-Header-Packet" '
		16#80005008 => 'MYSQL-ERROR: Unsupported value for "column count", provided as 24-bit value(3 bytes) in "Result-Set-Header-Packet" '
		16#80005009 => 'MYSQL-ERROR: Unsupported value for "column count", provided as 16-bit value(2 bytes) in "Result-Set-Header-Packet" '
		16#8000500A => 'MYSQL-ERROR: Length of identifier in column "x" exceed maximum of 250 bytes' 
		16#8000500B => 'MYSQL-ERROR: Identifier for "fieldname" in column "x" exceed maximum of "gcMySql_dwMaxIdentifierLength"';
		16#8000500C => 'MYSQL-ERROR: Length of row data exceed maximum of "gcMySql_dwMaxRowSize"
		16#8000500D => 'MYSQL-WARNING: Number of received rows exceed maximum of "gcMySql_dwMaxRowCount" - Some rows are ignored'
		16#80004001 => 'TIMEOUT: <actual processed step in state machine>'

	Remarks for "asSqlStatement":
	You can modify the "length" and number of elements in "asSqlStatement" by hiding 
	libraries global constants with global constants of same name in your project:
		- gcMySql_iSqlUpperBound:
				Defines the UpperBound of "asSqlStatement", to provide an SQL statement 
				as "ARRAY [0..UpperBound] OF STRING(Size)" 
		- gcMySql_iSqlLength:
				Defines the Size in byte of an array element of "asSqlStatement", 
				to provide an SQL statement as "ARRAY [0..UpperBound] OF STRING(Size)".   

	All non numeric SQL param values must be "quoted" with an apostroph(').
	Apostroph(') is also CoDesys-String-Start-End-Identifier.
	To use an apostroph(') inside a CoDeSys-String type $27 or $'.

	Example: 
		(* Prepare SQL-SELECT-Statement *)	
		asSqlStatement1[0] := 'SELECT * ';	
		asSqlStatement1[1] := 'FROM tablename ';	
		asSqlStatement1[2] := 'WHERE ';	
		asSqlStatement1[3] := ' name = $27Meyer$27 ';	
		asSqlStatement1[4] := ''; 						(* End of SQL-Statement *)

	Restriction: 
		- Maximum length for identifiers are 250 bytes!
		- Maximum length for field data are 500 bytes (TEXT, VARCHAR, ..!

 date     | release	| author  | Desc
----------+---------+------------------------------------------------------------
 21.03.14 |  3.8    | CM      | New "gcMySql_tResponseCompliedlyReceived"
 13.03.14 |  3.7	| CM      | Initialisation of "stResultSet" now optional("gcMySql_xClearResultSetBeforeUse := TRUE;" for debug purpose			
 02.07.12 |  3.6	| CM      | BugFix for large SQL-Statements 
 17.04.12 |  3.5	| CM      | BugFix for TIMEOUT error by "CALL <stored proc>"   
 24.01.12 |  3.4	| CM      | Bugfix for christmas tree on large error response
 26.09.11 |  3.3	| CM      | Clear complied "stResultSet" before use 
 16.09.11 |  3.2	| CM      | BugFix for large result sets 
 09.11.10 |  3.0    | CM      | Optimize cycletime, "stResultSet" now VAR_IN_OUT prior VAR_OUTPUT  
 19.08.10 |  2.1    | CM      | ReceiveBuffer handling modified to use full receive buffer 
 06.08.10 |  2.0	| CM      | Init 
*)
VAR_INPUT
	asSqlCommand : ARRAY [0..gcMySql_iSqlUpperBound] OF STRING(gcMySql_iSqlLength);
END_VAR
VAR_IN_OUT
	oMySql : MySql_Context; (* Structure for keeping login and status informations *)
	xStart : BOOL; 			(* Start execution on a rising edge and reseted internally when done or on timeout.  *)
	stResultSet : MySql_ResultSet; (* Query response data *)
END_VAR
VAR_OUTPUT
	diError : DWORD; 		(* Numeric return value - more readable in hex  *)
	sStatus : STRING(200); 	(* Textual description of current state or error *)
END_VAR
VAR
	wState : WORD;	 (* State mashine *)

	oTON			: TON;		(* Watchdogtimer for statemashine *)

	xWatchDogOn		: BOOL; 	(* enable disable Watchdog for statemashine *)
	wStateOld		: WORD;		(* persist the last state of statemashine *)

	xSemaOccupied	: BOOL;		(* This function block instance is current owner of critical path *)

	xResult			: BOOL;		(* Return value of functions *)
	diResult		: __XINT; 	(* Retval value of functions *)

	diTxCount		: __XINT; (* Number of bytes to send *)
	pbTxBufferPos	: POINTER TO BYTE; (* Position in Tx buffer of next data to transmit *)
	oTonTxDelay 	: TON; (* Delay for transmitting the rest package *)

	diRxCount		: __XINT; (* Number of received bytes within one TCP-Fragment *)
	diRxCountTotal  : __XINT; (* Total number of bytes received *)
	oTonRx			: TON;  (* Receive timeout, Go ahead if no new data received within the last 500ms *)

	(* Helpers *)
	dwPacketLength : DWORD; (*  *)
	uiPos : UINT;
	uiSubPos : UINT; (* *)

	dwMask : DWORD := 16#000000FF;
	uiCurrentField : UINT;
	uiCurrentRow : UINT;

	i,k : INT;
	iHelp : INT;
	diHelp : DINT;
	pabHelp : POINTER TO ARRAY [0..512] OF BYTE;
	RTS_IEC_RES: UDINT;
	ptrDINT : POINTER TO DINT;
END_VAR

CASE  wState OF (* The state maschine *********************************************)

0:	(* Idle - wait for something to do -------------------------------------------*)
	IF xStart THEN
		diError := 0;
		IF gcMySql_xClearResultSetBeforeUse THEN
			wState:=5; (* Clear "stResultSet" before use *)
		ELSE
			wState:=10; (* skip clearing of "stResultSet" *)
		END_IF
	END_IF

5: (* Clear "stResultSet" *)
	stResultSet.uiColumnCount := 0;
	FOR i:=0 TO DWORD_TO_INT(gcMySql_dwMaxColumnCount) DO
		stResultSet.astColumns[i].sName := 'UNUSED';
		stResultSet.astColumns[i].udiLength := 0;
		stResultSet.astColumns[i].eType := 0;
		stResultSet.astColumns[i].wFlags := 16#0000;
		stResultSet.astColumns[i].bDecimals := 16#00;
	END_FOR
	stResultSet.uiRowCount := 0;
	FOR i:=0 TO DWORD_TO_INT(gcMySql_dwMaxRowCount) DO
		FOR k:=0 TO DWORD_TO_INT(gcMySql_dwMaxRowSize) DO
			stResultSet.abRows[i][k] :=16#00;
		END_FOR
	END_FOR
	wState:=10; (* Go ahead *)

10: (* Check database connection --------------------------------------------------*)
	IF oMySql.xConnected THEN
		wState:=15; (* Go ahead *)
	ELSE
		diError := 16#80005005;
		sStatus :='MYSQL-ERROR: Not connected with database, LOGIN before use';
		wState:=999;
	END_IF

15: (* Wait until semaphore for Rx- and Tx-Buffer synchronization is available.
	With SysSemTry (which always returns immediately), a semaphore will be marked as used. 
	The returnvalue is TRUE if this succeeded and FALSE if the semaphore is already used by another task.  *)
	sStatus := 'Wait for semaphor';
	
	RTS_IEC_RES := SysSemTry(oMySql.dwBufferSemaphor);
	xResult := (RTS_IEC_RES = 0);
	IF xResult THEN
		xSemaOccupied := TRUE;
		sStatus := 'Execute SQL command';
		wState:=20; (* Go ahead *)
	END_IF

20: (*Prepare command packet "COM_QUERY"  ----------------------------------------*)
	(* Packet-Length - will be calculated and assigned at the end of this step *)
	oMySql.abTxBuffer[ 0] := 16#00;
	oMySql.abTxBuffer[ 1] := 16#00;
	oMySql.abTxBuffer[ 2] := 16#00;
	(* Packet-Number *)
	oMySql.abTxBuffer[ 3] := 0;
	(* Command-Type *)
	oMySql.abTxBuffer[ 4] := 16#03;  (* COM_QUERY - mysql_real_query *)
	(* Command-Argument (Null-Terminated String)*)
	uiPos := 5;
	FOR k:=0 TO gcMySql_iSqlUpperBound DO
		IF asSqlCommand[k] <> '' THEN
			pabHelp := ADR(asSqlCommand[k]);
			iHelp := LEN(asSqlCommand[k]);
			FOR i:=0 TO iHelp-1 DO
				oMySql.abTxBuffer[uiPos+i] := pabHelp^[i];
			END_FOR
			uiPos := uiPos + iHelp;
		ELSE
			EXIT;
		END_IF
	END_FOR
	oMySql.abTxBuffer[uiPos] := 16#00; (* Append STRING_END character "/0" *)
	uiPos := uiPos +1;
	(* Calculate number of bytes to transmit and logical packet-length *)
	diTxCount := uiPos; (* Bytes to send *)
	dwPacketLength := uiPos -4;
	(* Packet-Length *)
	oMySql.abTxBuffer[ 0] := DWORD_TO_BYTE(dwPacketLength AND dwMask);
	oMySql.abTxBuffer[ 1] := DWORD_TO_BYTE(SHR(dwPacketLength, 8) AND dwMask);
	oMySql.abTxBuffer[ 2] := DWORD_TO_BYTE(SHR(dwPacketLength, 16) AND dwMask);
	(* Set TxBufferPointer to begin of abTxBuffer *)
	pbTxBufferPos := ADR(oMySql.abTxBuffer);
	wState:=25; (* Go ahead *)

25: (* Send command packet "COM_QUERY"  ---------------------------*)
	diResult := SysSockSend(	hSocket := oMySql.dwSocketHandle,
								pbyBuffer := pbTxBufferPos,
								diBufferSize := diTxCount,
								diFlags := 0,
								pResult := ADR(RTS_IEC_RES));

	CASE diResult OF
	-1:	(* ERROR *)
		diError := 16#80001007;
		sStatus :='TCP-ERROR: "SysSockSend()" returns -1';
		wState:=999;
	0: (* Socket was "gracefully closed" *)
		MySql_Close(oMySql);
		diError := 16#80001006;
		sStatus :='TCP-ERROR: "SysSockSend()" returns 0. Socket was "gracefully closed"';
		wState:=999;
	ELSE (* succesful *)
		IF diResult >= diTxCount THEN
			(* All data transmitted *)
			diRxCountTotal := 0; (* Reset total number of bytes received *)
			wState:=30;
		ELSE
			(* Wait 200ms and then try to send the rest *)
			diTxCount := diTxCount - diResult;
			ptrDINT := ADR(diResult);
			pbTxBufferPos := pbTxBufferPos + ptrDINT^;
			wState:=27;
		END_IF
	END_CASE

27: (* Wait max ACK time (200ms) before send the rest, to support very slow servers also.
	   Function SysSockSend() will return -1 (Window Full) when you try to send the next 
	   package, before the last package are "ACKnoledged" by peer. *)
	oTonTxDelay(IN:=TRUE , PT:= t#200ms );
	IF oTonTxDelay.Q THEN
		oTonTxDelay(IN:=FALSE);
		wState := 25;
	END_IF

30: (* Wait for "Response" packets *)
	ptrDINT := ADR(diRxCountTotal);
	diHelp := SIZEOF(oMySql.abRxBuffer)-ptrDINT^; (* Calculate the free space of receive buffer *)
	(* Check if receive buffer able to store a complied tcp packet of 1460 bytes *)
	IF diHelp >= 1500 THEN
		(* Read from socket *)
		(*diRxCount := SysSockRecv(diSocket 	:= ,
								 pbyBuffer 	:= ADR(),	(* Address of receive buffer *)
								 diBufferSize:= ,			(* Maximum number of bytes to receive *)
								 diFlags	:= 0);*)
		diRxCount := SysSockRecv(		hSocket 	:= oMySql.dwSocketHandle,
										pbyBuffer 	:= ADR(oMySql.abRxBuffer[diRxCountTotal]),		(* Address of receive buffer *)
										diBufferSize:= diHelp,
										diFlags		:= 0,
										pResult := ADR(RTS_IEC_RES));						 

		CASE diRxCount OF
		-1:(* No data available or error occured *)
			IF diRxCountTotal = 0 THEN
				; (* Let the watchdog look for no response from server *)
			ELSE
				(* We have allready received some data, wait for more data to be shure complied response are received *)
				oTonRx(IN:=TRUE, PT:=gcMySql_tResponseCompliedlyReceived);
				IF oTonRx.Q THEN
					wState:=40; (* Go ahead *)
				END_IF
			END_IF

		(*0: (* Socket was "gracefully closed"  *)*)
			MySql_Close(oMySql);
			diError := 16#80001005;
			sStatus :='TCP-ERROR: "SysSockRecv()" returns 0. Socket was "gracefully closed"';
			wState:=999;
	
		ELSE (* We receive some data from server *)
			IF RTS_IEC_RES <> 0 AND RTS_IEC_RES <> 518 THEN
			diError := 16#80001005;
			sStatus :='TCP-ERROR: "SysSockRecv()" returns 0. Socket was "gracefully closed"';
			wState:=999;
		ELSE
		IF diRxCount > 0 THEN
			oTonRx(IN:=FALSE);
			diRxCountTotal := diRxCountTotal + diRxCount;
			(*Check if complied response are received, inicated by "EOF-Packet" *)
			IF oMySql.abRxBuffer[diRxCountTotal -5] = 16#FE THEN
				(* Last packet found *)
				wState:=40; (* Go ahead *)
			END_IF
		END_IF
		END_IF
		END_CASE
	ELSE
		MySql_Close(oMySql);
		diError := 16#80001008;
		sStatus :='TCP-ERROR: Receive buffer to small - increase "gcMySql_dwRxBufferSize"';
		wState:=999;
	END_IF

40: (* Check first response packet, could be a "Result-Set-Header-Packet" or "ERROR-Packet" *)
	uiPos := 0;
	dwPacketLength := 	BYTE_TO_DWORD(oMySql.abRxBuffer[uiPos]) OR
						SHL(BYTE_TO_DWORD(oMySql.abRxBuffer[uiPos+1]),8) OR
						SHL(BYTE_TO_DWORD(oMySql.abRxBuffer[uiPos+2]),16);
	(* Check Packet-Type *)
	CASE oMySql.abRxBuffer[uiPos+4] OF

	16#00:(* Invalid or unexpected response Packet-Type received from server (at this time) *)
		diError := 16#80005003;
		sStatus :='MYSQL-ERROR: Invalid or unexpected response from server';
		wState:=999;

	16#FF: (* ERROR-Packet: Identified by "field_count", always = 16#FF *)
		diError := 16#80005002;
		(* Copy server message into "sStatus"*)
		sStatus :='MYSQL-ERROR:  ';
		pabHelp := ADR(sStatus)+13;
		FOR i:=0 TO DWORD_TO_INT(dwPacketLength-10) DO
			pabHelp^[i] := oMySql.abRxBuffer[13+i];
			IF i>=180 THEN
				EXIT;
			END_IF
		END_FOR
		pabHelp^[i] := 16#00;
		wState:=999;

	16#FE: (* Value of "column count" are stored in following 64-bit (8 bytes) *)
		diError := 16#80005007;
		sStatus :='MYSQL-ERROR: Unsupported value for "column count", provided as 64-bit value(8 bytes) in "Result-Set-Header-Packet" ';
		wState:=999;

	16#FD: (* Value of "column count" are stored in following 24-bit (3 bytes) *)
		diError := 16#80005008;
		sStatus :='MYSQL-ERROR: Unsupported value for "column count", provided as 24-bit value(3 bytes) in "Result-Set-Header-Packet" ';
		wState:=999;

	16#FC: (* Value of "column count" are stored in following 16-bit (2 bytes) *)
		diError := 16#80005009;
		sStatus :='MYSQL-ERROR: Unsupported value for "column count", provided as 16-bit value(2 bytes) in "Result-Set-Header-Packet" ';
		wState:=999;

	16#FB: (* column value = NULL - only appropriate in a Row Data Packet, so unexpected here *)
		diError := 16#80005003;
		sStatus :='MYSQL-ERROR: Invalid or unexpected response packet from server';
		wState:=999;

	ELSE
		(* Read "column count", the number of columns in result set - (length coded binary) *)
		stResultSet.uiColumnCount := BYTE_TO_UINT(oMySql.abRxBuffer[uiPos+4]);
		uiPos := 5;
		(* Check column count against maximum *)
		IF stResultSet.uiColumnCount <= gcMySql_dwMaxColumnCount THEN
			uiCurrentField :=0; (* Init *)
			wState:=50;
		ELSE
			diError := 16#80005006;
			sStatus :='MYSQL-ERROR: Result set has more columns then defined in "gcMySql_dwMaxColumnCount"';
			wState:=999;
		END_IF

	END_CASE

50: (* Process next response packets, must be a "Field-Packet" *)
	dwPacketLength := 	BYTE_TO_DWORD(oMySql.abRxBuffer[uiPos]) OR
						SHL(BYTE_TO_DWORD(oMySql.abRxBuffer[uiPos+1]),8) OR
						SHL(BYTE_TO_DWORD(oMySql.abRxBuffer[uiPos+2]),16);
	uiSubPos := uiPos +4;
	(* Iterate over field informations: "catalog", "db", "table", "org_table", "name", "org_name" *)
	FOR i:=0 TO 5 DO
		(* Check length information (Binary coded length *)
		IF oMySql.abRxBuffer[uiSubPos] <= 250 THEN
			IF i=4 THEN (* Copy "name" *)
				IF oMySql.abRxBuffer[uiSubPos] <= gcMySql_dwMaxIdentifierLength  THEN
					pabHelp := ADR(stResultSet.astColumns[uiCurrentField].sName);
					FOR k:=0 TO oMySql.abRxBuffer[uiSubPos] -1 DO
						pabHelp^[k] := oMySql.abRxBuffer[uiSubPos+1+k];
					END_FOR
					pabHelp^[k] := 16#00; (* Append String end "\0" *)
				ELSE
					diError := 16#8000500B;
					sStatus :=CONCAT('MYSQL-ERROR: Identifier for "fieldname" in column "', UINT_TO_STRING(uiCurrentField+1));
					sStatus :=CONCAT(sStatus, '" exceed maximum of ');
					sStatus :=CONCAT(sStatus, DWORD_TO_STRING(gcMySql_dwMaxIdentifierLength));
					wState:=999;
					RETURN; (***** RETURN *****)
				END_IF
			END_IF
			uiSubPos := uiSubPos + oMySql.abRxBuffer[uiSubPos]+1;
		ELSE
			diError := 16#8000500A;
			sStatus :=CONCAT('MYSQL-ERROR: Length of identifier in column "', UINT_TO_STRING(uiCurrentField+1));
			sStatus :=CONCAT(sStatus, '" exceed maximum of 250 bytes');
			wState:=999;
			RETURN; (***** RETURN *****)
		END_IF
	END_FOR
	uiSubPos := uiSubPos + 3; (* Skip "filler" and "charsetnumber" *)
	(* Copy "length" *)
	stResultSet.astColumns[uiCurrentField].udiLength := DWORD_TO_UDINT(
					BYTE_TO_DWORD(oMySql.abRxBuffer[uiSubPos  ]) 		OR
				SHL(BYTE_TO_DWORD(oMySql.abRxBuffer[uiSubPos+1]),8) 	OR
				SHL(BYTE_TO_DWORD(oMySql.abRxBuffer[uiSubPos+2]),16)    OR
				SHL(BYTE_TO_DWORD(oMySql.abRxBuffer[uiSubPos+3]),24)
				);
	uiSubPos := uiSubPos + 4;
	(* Copy "type" *)
	stResultSet.astColumns[uiCurrentField].eType := oMySql.abRxBuffer[uiSubPos];
	uiSubPos := uiSubPos + 1;
	(* Copy "flags" *)
	stResultSet.astColumns[uiCurrentField].wFlags := BYTE_TO_WORD(oMySql.abRxBuffer[uiSubPos  ]) 		OR
												 SHL(BYTE_TO_WORD(oMySql.abRxBuffer[uiSubPos+1]),8);
	uiSubPos := uiSubPos + 2;
	(* Copy "decimals" *)
	stResultSet.astColumns[uiCurrentField].bDecimals :=  oMySql.abRxBuffer[uiSubPos];

	(* Set read position in receive buffer to head of next  "Field-Packet"  *)
	uiPos := uiPos + DWORD_TO_UINT(dwPacketLength) +4;
	uiCurrentField := uiCurrentField +1; (* Increment processed "Field-Packet's"*)
	IF uiCurrentField >= stResultSet.uiColumnCount THEN
		wState:=60;
	END_IF;

60: (* Process next response packets, must be a "EOF-Packet" *)
	dwPacketLength := 	BYTE_TO_DWORD(oMySql.abRxBuffer[uiPos]) OR
						SHL(BYTE_TO_DWORD(oMySql.abRxBuffer[uiPos+1]),8) OR
						SHL(BYTE_TO_DWORD(oMySql.abRxBuffer[uiPos+2]),16);
	(* Check Packet-Type *)
	IF oMySql.abRxBuffer[uiPos+4] = 16#FE THEN
		(* Set read position in receive buffer to head of next packet *)
		uiPos := uiPos + DWORD_TO_UINT(dwPacketLength) +4;
		uiCurrentRow := 0; (* Init row counter *)
		wState:=70;
	ELSE
		diError := 16#80005003;
		sStatus :='MYSQL-ERROR: Invalid or unexpected response from server';
		wState:=999;
	END_IF

70: (* Process "Row-Data-Packets" until find "EOF-Packet" *)
	dwPacketLength := 	BYTE_TO_DWORD(oMySql.abRxBuffer[uiPos]) OR
						SHL(BYTE_TO_DWORD(oMySql.abRxBuffer[uiPos+1]),8) OR
						SHL(BYTE_TO_DWORD(oMySql.abRxBuffer[uiPos+2]),16);
	(* Check if current packet is a "EOF-Packet" or "Row-Data-Packet" *)
	IF oMySql.abRxBuffer[uiPos+4] = 16#FE THEN
		(* Packet type is "EOF-Packet" - No more data in this packet *)
		stResultSet.uiRowCount := uiCurrentRow;
		sStatus := CONCAT('Successful executed - affected rows: ', UINT_TO_STRING(stResultSet.uiRowCount));
		(* Check servers "Status-Flags" for all data received *)
		IF (oMySql.abRxBuffer[uiPos+7] AND 16#40) > 0 THEN
			(* More rows available on server  *)
			sStatus := CONCAT(sStatus, ' - More rows available on server !!!! ');
		END_IF
		wState:=999;
	ELSE
		(* Packet type is "Row-Data-Packet" - Copy data into "stResultSet" *)
		IF uiCurrentRow < gcMySql_dwMaxRowCount THEN
			IF dwPacketLength <= gcMySql_dwMaxRowSize THEN
				FOR i:=0 TO DWORD_TO_INT(dwPacketLength -1) DO
					stResultSet.abRows[uiCurrentRow][i] := oMySql.abRxBuffer[uiPos+4+i];
				END_FOR
				stResultSet.abRows[uiCurrentRow][i] := 16#00; (* Append String end "\0" (New in version 3.7)*)
				(* Set read position in receive buffer to head of next packet *)
				uiPos := uiPos + DWORD_TO_UINT(dwPacketLength) +4;
				uiCurrentRow := uiCurrentRow +1; (* Increment internal row counter *)
				stResultSet.uiRowCount := uiCurrentRow; (* Update "stResultSet" *)
			ELSE
				diError := 16#8000500C;
				sStatus :='MYSQL-ERROR: Length of row data exceed maximum of "gcMySql_dwMaxRowSize"';
				wState:=999;
				RETURN; (***** RETURN *****)
			END_IF
		ELSE
			diError := 16#8000500D;
			sStatus :='MYSQL-WARNING: Number of received rows exceed maximum of "gcMySql_dwMaxRowCount" - Some rows are ignored';
			wState:=999;
			RETURN; (***** RETURN *****)
		END_IF
	END_IF

ELSE
	(* Clean up and leave connection open -----------------------------------------*)
	IF xSemaOccupied THEN
		SysSemLeave(oMySql.dwBufferSemaphor); (* Leave semaphore, to be shure nowbody is blocked by her *)
		xSemaOccupied := FALSE;
	END_IF
	xStart := FALSE;
	wState:=0;

END_CASE (**************************************************************************************)


(* Watchdog for statemachine  *)
IF oTON.Q THEN
	xWatchDogOn := FALSE;
	diError := 16#80004001; 	(* Watchdog time elapsed, see sStatus for details *)
	sStatus := CONCAT('TIMEOUT on:', sStatus);
	wState:=999;
END_IF

IF (wState > 0) THEN
	oTON(IN:=xWatchDogOn , PT:=gcMySql_tTimeOut);
	IF (wStateOld <> wState) THEN
		xWatchDogOn := FALSE; (* Step has changed *)
	ELSE
		xWatchDogOn := TRUE; (* Step still active *)
	END_IF
END_IF
wStateOld:=wState;

END_FUNCTION_BLOCK

// Device/Application/Cycletime
FUNCTION_BLOCK Cycletime

VAR
	clock_up: UDINT;
END_VAR
VAR // added by the converter: edge detectors and wires of the graphical bodies
    _rt1, _rt2 : R_TRIG;
END_VAR

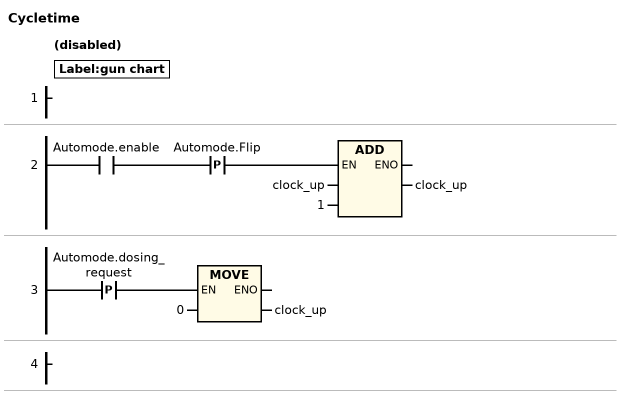
// NETWORK 1 (disabled)
// label: Label:gun chart

// NETWORK 2
_rt1(CLK := Automode.Flip);
IF Automode.enable AND _rt1.Q THEN clock_up := clock_up + 1; END_IF

// NETWORK 3
_rt2(CLK := Automode.dosing_request);
IF _rt2.Q THEN clock_up := 0; END_IF

// NETWORK 4

END_FUNCTION_BLOCK

// Device/Application/MYSQL/private/SHA/SHA1Version
FUNCTION SHA1Version : WORD
(*
*  Copyright (C) 1998, 2009
*  Paul E. Jones <paulej@packetizer.com>
*  All Rights Reserved
*
*****************************************************************************
*  $Id: sha1.h 12 2009-06-22 19:34:25Z paulej $
*****************************************************************************
*
*  Description:
*      This class implements the Secure Hashing Standard as defined
*      in FIPS PUB 180-1 published April 17, 1995.
*
*      Many of the variable names in the SHA1Context, especially the
*      single character names, were used because those were the names
*      used in the publication.
*

 date     | release	| author  | Desc
----------+---------+------------------------------------------------------------
 08.03.11 |  1.2	| CM      | Add some comments, no functional change
 02.08.10 |  1.1	| CM      | Add param "pabDigest" to function "SHA1Result"   
 20.07.10 |  1.0	| CM      | Port to IEC 6-1131 
 22.06.09 |  0.0	| PEJ     | Original (C-Code)  
 
 *)
VAR_INPUT
END_VAR
VAR
	(* Current library version *)
	bMajor : BYTE := 16#01;
	bMinor : BYTE := 16#02;
END_VAR

SHA1Version := SHL(BYTE_TO_WORD(bMajor), 8) OR BYTE_TO_WORD(bMinor);

END_FUNCTION

// Device/Application/MYSQL/public/MySql_GetStringValue
FUNCTION MySql_GetStringValue : DWORD
(* This function convert the requested field data into a IEC61131 data type and returns it as string.

	RetVal 	
		16#00000000 => 'SUCCESS'
		16#80006001 => 'PARAM-ERROR: Invalid param "row" - First row start on index 1. ;
		16#80006002 => 'PARAM-ERROR: Invalid param "col" - First col start on index 1. ;
		16#80006003 => 'PARAM-ERROR: Requested row do not exist in "stQueryResult";
		16#80006004 => 'PARAM-ERROR: Requested col do not exist in "stQueryResult";
		16#80006005 => 'CONVERT-ERROR: Length of col "x" exceed maximum of 500 bytes;
		16#80006006 => 'CONVERT-ERROR: Field "x" use unsupported 8byte style for length informations';
		16#80006007 => 'CONVERT-ERROR: Unknown MySQL-Data-Type: "x"';
		16#80006008 => 'CONVERT-ERROR: Unsupported MySQL-Data-Type: "x"';

	ToDo:
		- Enable large fields (currently limited to 500 bytes) 

 date     | release	| author  | Desc
----------+---------+------------------------------------------------------------
 06.12.10 |  3.1    | CM      | BugFix for Fieldtype 'TOD#'
 06.08.10 |  2.0	| CM      | Init 

*)
VAR_INPUT
	iRow : INT; 	(* Row to process, start with index 1 for the first row *)
	iCol : INT; 	(* Column to process, start with index 1 for the first column  *)
END_VAR
VAR_IN_OUT
	stQueryResult : MySql_ResultSet;
	sValue: STRING(500); 	(* Value as STRING(500) or error message *)
END_VAR
VAR
	uiPos : UINT; 			(* Position in actual row *)
	uiLength : UINT;
	iCurrentCol : INT; 		(* Actual column to process *)
	abHelp : ARRAY [0..512] OF BYTE; (* Buffer for syntax modification *)
	psHelp : POINTER TO STRING(500); (* Helper for type cast *)
	i : INT;
END_VAR

(* Check param "row" *)
IF iRow =0 THEN
	sValue := 'PARAM-ERROR: Invalid param "row" - First row start on index 1';
	MySql_GetStringValue := 16#80006001;
	RETURN;
END_IF
(* Check param "col" *)
IF iCol = 0 THEN
	sValue := 'PARAM-ERROR: Invalid param "col" - First col start on index 1';
	MySql_GetStringValue := 16#80006002;
	RETURN;
END_IF
(* Check requested "row" for valid value *)
IF iRow > stQueryResult.uiRowCount THEN
	sValue := 'PARAM-ERROR: Requested row do not exist in "stQueryResult"';
	MySql_GetStringValue := 16#80006003;
	RETURN;
END_IF
(* Check requested "col" for valid value *)
IF iCol > stQueryResult.uiColumnCount THEN
	sValue := 'CONVERT-ERROR: Requested column do not exist in "stQueryResult"';
	MySql_GetStringValue := 16#80006004;
	RETURN;
END_IF

iCurrentCol := 0;
uiPos := 0;
(* Find position of requested field and get the length of it *)
REPEAT
	CASE stQueryResult.abRows[iRow-1][uiPos] OF
	251: (* column value = "NULL" only appropriate in a "Row-Data-Packet" *)
		uiLength := 0;
		uiPos := uiPos +1;
		sValue := 'NULL';
	252: (* Length defined by following two bytes(Value of following 16-bit) *)
		uiLength := DWORD_TO_UINT(  BYTE_TO_DWORD(stQueryResult.abRows[iRow-1][uiPos]) OR
								SHL(BYTE_TO_DWORD(stQueryResult.abRows[iRow-1][uiPos+1]),8) );
		sValue := '';
		uiPos := uiPos +3;

	253: (* Length defined by following three bytes(Value of following 24-bit) *)
		uiLength := DWORD_TO_UINT(  BYTE_TO_DWORD(stQueryResult.abRows[iRow-1][uiPos]) OR
								SHL(BYTE_TO_DWORD(stQueryResult.abRows[iRow-1][uiPos+1]),8) OR
								SHL(BYTE_TO_DWORD(stQueryResult.abRows[iRow-1][uiPos+2]),16));
		sValue := '';
		uiPos := uiPos +4;

	254: (* Length defined by following 8 bytes(Value of following 64-bit) *)
		uiLength := 0;
		sValue := CONCAT('CONVERT-ERROR: Field "', INT_TO_STRING(i));
		sValue := CONCAT(sValue, '" use unsupported 8byte style for length information');
		MySql_GetStringValue := 16#80006006;
		RETURN;

	ELSE
		(* Length is between 0..250 bytes *)
		uiLength := stQueryResult.abRows[iRow-1][uiPos];
		sValue := '';
		uiPos := uiPos +1;
	END_CASE
	iCurrentCol := iCurrentCol +1;

	(* Check if current col is the requested col *)
	IF (iCurrentCol = iCol) THEN
		(* Convert and copy field data into "sValue" *)
		EXIT;
	ELSE
		(* Skip to next column *)
		IF sValue = '' THEN  (* "sValue = '' indicate that uiPos points to the begin of field data *)
			uiPos := uiPos +uiLength;
		END_IF
	END_IF

UNTIL (iCurrentCol >= iCol)
END_REPEAT

(* Check if sValue contains an error message or not *)
IF sValue = '' THEN (* "sValue = '' indicate that "uiPos" points to the begin of field data *)
	(* Convert and copy field content into "sValue" depended of its MySQL-Data-Type *)
	CASE stQueryResult.astColumns[iCol-1].eType OF
		(* Integers *)
		MYSQL_TYPE_TINY,
		MYSQL_TYPE_SHORT,
		MYSQL_TYPE_LONG,
		MYSQL_TYPE_INT24,
		MYSQL_TYPE_LONGLONG,
		(* char fields *)
		MYSQL_TYPE_VAR_STRING,
		MYSQL_TYPE_STRING,
		MYSQL_TYPE_VARCHAR,
		(* Floating point types *)
		MYSQL_TYPE_DECIMAL,
		MYSQL_TYPE_NEWDECIMAL,
		MYSQL_TYPE_FLOAT,
		MYSQL_TYPE_DOUBLE: (* Just copy into buffer and append [EOF] *)
			FOR i:=0 TO uiLength-1 DO
				abHelp[ i] := stQueryResult.abRows[iRow-1][uiPos+i];
			END_FOR
			abHelp[i] := 16#00; (* [EOF] *)
			psHelp := ADR(abHelp);
			sValue := psHelp^;

		MYSQL_TYPE_DATETIME,
		MYSQL_TYPE_TIMESTAMP: (* Convert timestamp to DT-Format: 'dt#1970-01-01-00:00:00'  *)
			abHelp[ 0] := 16#64; (*  "d"  *)
			abHelp[ 1] := 16#74; (*  "t"  *)
			abHelp[ 2] := 16#23; (*  "#"  *)
			abHelp[ 3] := stQueryResult.abRows[iRow-1][uiPos   ];
			abHelp[ 4] := stQueryResult.abRows[iRow-1][uiPos+1 ];
			abHelp[ 5] := stQueryResult.abRows[iRow-1][uiPos+2 ];
			abHelp[ 6] := stQueryResult.abRows[iRow-1][uiPos+3 ];
			abHelp[ 7] := 16#2D; (*  "-"  *)
			abHelp[ 8] := stQueryResult.abRows[iRow-1][uiPos+5 ];
			abHelp[ 9] := stQueryResult.abRows[iRow-1][uiPos+6 ];
			abHelp[10] := 16#2D; (*  "-"  *)
			abHelp[11] := stQueryResult.abRows[iRow-1][uiPos+8 ];
			abHelp[12] := stQueryResult.abRows[iRow-1][uiPos+9 ];
			abHelp[13] := 16#2D; (*  "-"  *)
			abHelp[14] := stQueryResult.abRows[iRow-1][uiPos+11];
			abHelp[15] := stQueryResult.abRows[iRow-1][uiPos+12];
			abHelp[16] := 16#3A; (*  ":"  *)
			abHelp[17] := stQueryResult.abRows[iRow-1][uiPos+14];
			abHelp[18] := stQueryResult.abRows[iRow-1][uiPos+15];
			abHelp[19] := 16#3A; (*  ":"  *)
			abHelp[20] := stQueryResult.abRows[iRow-1][uiPos+17];
			abHelp[21] := stQueryResult.abRows[iRow-1][uiPos+18];
			abHelp[22] := 16#00; (* [EOF] *)
			psHelp := ADR(abHelp);
			sValue := psHelp^;

		MYSQL_TYPE_DATE: (* Convert date to D-Format: 'd#1970-01-01'  *)
			abHelp[ 0] := 16#64; (*  "d"  *)
			abHelp[ 1] := 16#23; (*  "#"  *)
			abHelp[ 2] := stQueryResult.abRows[iRow-1][uiPos   ];
			abHelp[ 3] := stQueryResult.abRows[iRow-1][uiPos+1 ];
			abHelp[ 4] := stQueryResult.abRows[iRow-1][uiPos+2 ];
			abHelp[ 5] := stQueryResult.abRows[iRow-1][uiPos+3 ];
			abHelp[ 6] := 16#2D; (*  "-"  *)
			abHelp[ 7] := stQueryResult.abRows[iRow-1][uiPos+5 ];
			abHelp[ 8] := stQueryResult.abRows[iRow-1][uiPos+6 ];
			abHelp[ 9] := 16#2D; (*  "-"  *)
			abHelp[10] := stQueryResult.abRows[iRow-1][uiPos+8 ];
			abHelp[11] := stQueryResult.abRows[iRow-1][uiPos+9 ];
			abHelp[12] := 16#00; (* [EOF] *)
			psHelp := ADR(abHelp);
			sValue := psHelp^;

		MYSQL_TYPE_TIME: (* Convert time to TOD-Format: 'tod#00:00:00'  *)
			abHelp[ 0] := 16#74; (*  "t"  *)
			abHelp[ 1] := 16#6F; (*  "o"  *)
			abHelp[ 2] := 16#64; (*  "d"  *)
			abHelp[ 3] := 16#23; (*  "#"  *)
			abHelp[ 4] := stQueryResult.abRows[iRow-1][uiPos];
			abHelp[ 5] := stQueryResult.abRows[iRow-1][uiPos+1];
			abHelp[ 6] := 16#3A; (*  ":"  *)
			abHelp[ 7] := stQueryResult.abRows[iRow-1][uiPos+3];
			abHelp[ 8] := stQueryResult.abRows[iRow-1][uiPos+4];
			abHelp[ 9] := 16#3A; (*  ":"  *)
			abHelp[10] := stQueryResult.abRows[iRow-1][uiPos+6];
			abHelp[11] := stQueryResult.abRows[iRow-1][uiPos+7];
			abHelp[12] := 16#00; (* [EOF] *)
			psHelp := ADR(abHelp);
			sValue := psHelp^;


